GVL.arrValve_PM[0](in_out:= GVL.pm[0].inConv.valve[0]);
GVL.arrValve_PM[1](in_out:= GVL.pm[0].inConv.valve[1]);
GVL.arrValve_PM[2](in_out:= GVL.pm[0].inConv.valve[2]);
GVL.arrValve_PM[3](in_out:= GVL.pm[1].inConv.valve[0]);
GVL.arrValve_PM[4](in_out:= GVL.pm[1].inConv.valve[1]);
GVL.arrValve_PM[5](in_out:= GVL.pm[1].inConv.valve[2]);
GVL.arrValve_PM[6](in_out:= GVL.pm[2].inConv.valve[0]);
GVL.arrValve_PM[7](in_out:= GVL.pm[2].inConv.valve[1]);
GVL.arrValve_PM[8](in_out:= GVL.pm[2].inConv.valve[2]);
GVL.arrValve_PM[9](in_out:= GVL.pm[3].inConv.valve[0]);
GVL.arrValve_PM[10](in_out:= GVL.pm[3].inConv.valve[1]);
GVL.arrValve_PM[11](in_out:= GVL.pm[3].inConv.valve[2]);
GVL.arrValve_PM[12](in_out:= GVL.pm[4].inConv.valve[0]);
GVL.arrValve_PM[13](in_out:= GVL.pm[4].inConv.valve[1]);
GVL.arrValve_PM[14](in_out:= GVL.pm[4].inConv.valve[2]);
GVL.arrValve_PM[15](in_out:= GVL.pm[5].inConv.valve[0]);
GVL.arrValve_PM[16](in_out:= GVL.pm[5].inConv.valve[1]);
GVL.arrValve_PM[17](in_out:= GVL.pm[5].inConv.valve[2]);
GVL.arrValve_PM[18](in_out:= GVL.pm[6].inConv.valve[0]);
GVL.arrValve_PM[19](in_out:= GVL.pm[6].inConv.valve[1]);
GVL.arrValve_PM[20](in_out:= GVL.pm[6].inConv.valve[2]);
GVL.arrValve_PM[21](in_out:= GVL.pm[7].inConv.valve[0]);
GVL.arrValve_PM[22](in_out:= GVL.pm[7].inConv.valve[1]);
GVL.arrValve_PM[23](in_out:= GVL.pm[7].inConv.valve[2]);
GVL.arrValve_PM[24](in_out:= GVL.pm[8].inConv.valve[0]);
GVL.arrValve_PM[25](in_out:= GVL.pm[8].inConv.valve[1]);
GVL.arrValve_PM[26](in_out:= GVL.pm[8].inConv.valve[2]);
GVL.arrValve_PM[27](in_out:= GVL.pm[9].inConv.valve[0]);
GVL.arrValve_PM[28](in_out:= GVL.pm[9].inConv.valve[1]);
GVL.arrValve_PM[29](in_out:= GVL.pm[9].inConv.valve[2]);
GVL.arrValve_PM[30](in_out:= GVL.pm[0].outConv.valve[0]);
GVL.arrValve_PM[31](in_out:= GVL.pm[0].outConv.valve[1]);
GVL.arrValve_PM[32](in_out:= GVL.pm[1].outConv.valve[0]);
GVL.arrValve_PM[33](in_out:= GVL.pm[1].outConv.valve[1]);
GVL.arrValve_PM[34](in_out:= GVL.pm[2].outConv.valve[0]);
GVL.arrValve_PM[35](in_out:= GVL.pm[2].outConv.valve[1]);
GVL.arrValve_PM[36](in_out:= GVL.pm[3].outConv.valve[0]);
GVL.arrValve_PM[37](in_out:= GVL.pm[3].outConv.valve[1]);
GVL.arrValve_PM[38](in_out:= GVL.pm[4].outConv.valve[0]);
GVL.arrValve_PM[39](in_out:= GVL.pm[4].outConv.valve[1]);
GVL.arrValve_PM[40](in_out:= GVL.pm[5].outConv.valve[0]);
GVL.arrValve_PM[41](in_out:= GVL.pm[5].outConv.valve[1]);
GVL.arrValve_PM[42](in_out:= GVL.pm[6].outConv.valve[0]);
GVL.arrValve_PM[43](in_out:= GVL.pm[6].outConv.valve[1]);
GVL.arrValve_PM[44](in_out:= GVL.pm[7].outConv.valve[0]);
GVL.arrValve_PM[45](in_out:= GVL.pm[7].outConv.valve[1]);
GVL.arrValve_PM[46](in_out:= GVL.pm[8].outConv.valve[0]);
GVL.arrValve_PM[47](in_out:= GVL.pm[8].outConv.valve[1]);
GVL.arrValve_PM[48](in_out:= GVL.pm[9].outConv.valve[0]);
GVL.arrValve_PM[49](in_out:= GVL.pm[9].outConv.valve[1]);//end of pm
GVL.arrValve_PM[50](in_out:= GVL.lb[0].valve_stopper[0]);
GVL.arrValve_PM[51](in_out:= GVL.lb[0].valve_stopper[1]);
GVL.arrValve_PM[52](in_out:= GVL.lb[0].valve_stopper[2]);
GVL.arrValve_PM[53](in_out:= GVL.lb[0].valve_stopper[3]);
GVL.arrValve_PM[54](in_out:= GVL.lb[0].valve_stopper[4]);
GVL.arrValve_PM[55](in_out:= GVL.lb[0].valve_stopper[5]);
GVL.arrValve_PM[56](in_out:= GVL.lb[1].valve_stopper[0]);
GVL.arrValve_PM[57](in_out:= GVL.lb[1].valve_stopper[1]);
GVL.arrValve_PM[58](in_out:= GVL.lb[1].valve_stopper[2]);
GVL.arrValve_PM[59](in_out:= GVL.lb[1].valve_stopper[3]);
GVL.arrValve_PM[60](in_out:= GVL.lb[1].valve_stopper[4]);
GVL.arrValve_PM[61](in_out:= GVL.lb[1].valve_stopper[5]);//end of lb
GVL.arrValve_PM[62](in_out:= GVL.lc[0].valve_guide[0]);
GVL.arrValve_PM[63](in_out:= GVL.lc[0].valve_guide[1]);
GVL.arrValve_PM[64](in_out:= GVL.lc[0].valve_stopper[0]);
GVL.arrValve_PM[65](in_out:= GVL.lc[0].valve_stopper[1]);
GVL.arrValve_PM[66](in_out:= GVL.lc[0].lateral.valve_lift);
GVL.arrValve_PM[67](in_out:= GVL.lc[0].lateral.valve_clamp[0]);
GVL.arrValve_PM[68](in_out:= GVL.lc[0].lateral.valve_clamp[1]);
GVL.arrValve_PM[69](in_out:= GVL.lc[1].valve_guide[0]);
GVL.arrValve_PM[70](in_out:= GVL.lc[1].valve_guide[1]);
GVL.arrValve_PM[71](in_out:= GVL.lc[1].valve_stopper[0]);
GVL.arrValve_PM[72](in_out:= GVL.lc[1].valve_stopper[1]);
GVL.arrValve_PM[73](in_out:= GVL.lc[1].lateral.valve_lift);
GVL.arrValve_PM[74](in_out:= GVL.lc[1].lateral.valve_clamp[0]);
GVL.arrValve_PM[75](in_out:= GVL.lc[1].lateral.valve_clamp[1]);//end of lc
GVL.arrValve_PM[76](in_out:= GVL.fr[0].valve);
GVL.arrValve_PM[77](in_out:= GVL.fr[1].valve);//end of fr

//////////////////////////////////////REM/////////////////////////////////////
GVL.arrValve_Rem[0](in_out:= GVL.rem[0].infeed[0].valve_stopper);
GVL.arrValve_Rem[1](in_out:= GVL.rem[0].lift[0].valve_clamp);
GVL.arrValve_Rem[2](in_out:= GVL.rem[0].lift[0].valve_perturbation[0]);
GVL.arrValve_Rem[3](in_out:= GVL.rem[0].lift[0].valve_perturbation[1]);
GVL.arrValve_Rem[4](in_out:= GVL.rem[0].lift[0].valve_perturbation[2]);
GVL.arrValve_Rem[5](in_out:= GVL.rem[0].lift[0].valve_perturbation[3]);
GVL.arrValve_Rem[6](in_out:= GVL.rem[0].infeed[1].valve_stopper);
GVL.arrValve_Rem[7](in_out:= GVL.rem[0].lift[1].valve_clamp);
GVL.arrValve_Rem[8](in_out:= GVL.rem[0].lift[1].valve_perturbation[0]);
GVL.arrValve_Rem[9](in_out:= GVL.rem[0].lift[1].valve_perturbation[1]);
GVL.arrValve_Rem[10](in_out:= GVL.rem[0].lift[1].valve_perturbation[2]);
GVL.arrValve_Rem[11](in_out:= GVL.rem[0].lift[1].valve_perturbation[3]);
GVL.arrValve_Rem[12](in_out:= GVL.rem[1].infeed[0].valve_stopper);
GVL.arrValve_Rem[13](in_out:= GVL.rem[1].lift[0].valve_clamp);
GVL.arrValve_Rem[14](in_out:= GVL.rem[1].lift[0].valve_perturbation[0]);
GVL.arrValve_Rem[15](in_out:= GVL.rem[1].lift[0].valve_perturbation[1]);
GVL.arrValve_Rem[16](in_out:= GVL.rem[1].lift[0].valve_perturbation[2]);
GVL.arrValve_Rem[17](in_out:= GVL.rem[1].lift[0].valve_perturbation[3]);
GVL.arrValve_Rem[18](in_out:= GVL.rem[1].infeed[1].valve_stopper);
GVL.arrValve_Rem[19](in_out:= GVL.rem[1].lift[1].valve_clamp);
GVL.arrValve_Rem[20](in_out:= GVL.rem[1].lift[1].valve_perturbation[0]);
GVL.arrValve_Rem[21](in_out:= GVL.rem[1].lift[1].valve_perturbation[1]);
GVL.arrValve_Rem[22](in_out:= GVL.rem[1].lift[1].valve_perturbation[2]);
GVL.arrValve_Rem[23](in_out:= GVL.rem[1].lift[1].valve_perturbation[3]);
GVL.arrValve_Rem[24](in_out:= GVL.rem[2].infeed[0].valve_stopper);
GVL.arrValve_Rem[25](in_out:= GVL.rem[2].lift[0].valve_clamp);
GVL.arrValve_Rem[26](in_out:= GVL.rem[2].lift[0].valve_perturbation[0]);
GVL.arrValve_Rem[27](in_out:= GVL.rem[2].lift[0].valve_perturbation[1]);
GVL.arrValve_Rem[28](in_out:= GVL.rem[2].lift[0].valve_perturbation[2]);
GVL.arrValve_Rem[29](in_out:= GVL.rem[2].lift[0].valve_perturbation[3]);
GVL.arrValve_Rem[30](in_out:= GVL.rem[2].infeed[1].valve_stopper);
GVL.arrValve_Rem[31](in_out:= GVL.rem[2].lift[1].valve_clamp);
GVL.arrValve_Rem[32](in_out:= GVL.rem[2].lift[1].valve_perturbation[0]);
GVL.arrValve_Rem[33](in_out:= GVL.rem[2].lift[1].valve_perturbation[1]);
GVL.arrValve_Rem[34](in_out:= GVL.rem[2].lift[1].valve_perturbation[2]);
GVL.arrValve_Rem[35](in_out:= GVL.rem[2].lift[1].valve_perturbation[3]);
GVL.arrValve_Rem[36](in_out:= GVL.rem[3].infeed[0].valve_stopper);
GVL.arrValve_Rem[37](in_out:= GVL.rem[3].lift[0].valve_clamp);
GVL.arrValve_Rem[38](in_out:= GVL.rem[3].lift[0].valve_perturbation[0]);
GVL.arrValve_Rem[39](in_out:= GVL.rem[3].lift[0].valve_perturbation[1]);
GVL.arrValve_Rem[40](in_out:= GVL.rem[3].lift[0].valve_perturbation[2]);
GVL.arrValve_Rem[41](in_out:= GVL.rem[3].lift[0].valve_perturbation[3]);
GVL.arrValve_Rem[42](in_out:= GVL.rem[3].infeed[1].valve_stopper);
GVL.arrValve_Rem[43](in_out:= GVL.rem[3].lift[1].valve_clamp);
GVL.arrValve_Rem[44](in_out:= GVL.rem[3].lift[1].valve_perturbation[0]);
GVL.arrValve_Rem[45](in_out:= GVL.rem[3].lift[1].valve_perturbation[1]);
GVL.arrValve_Rem[46](in_out:= GVL.rem[3].lift[1].valve_perturbation[2]);
GVL.arrValve_Rem[47](in_out:= GVL.rem[3].lift[1].valve_perturbation[3]);
GVL.arrValve_Rem[48](in_out:= GVL.rem[4].infeed[0].valve_stopper);
GVL.arrValve_Rem[49](in_out:= GVL.rem[4].lift[0].valve_clamp);
GVL.arrValve_Rem[50](in_out:= GVL.rem[4].lift[0].valve_perturbation[0]);
GVL.arrValve_Rem[51](in_out:= GVL.rem[4].lift[0].valve_perturbation[1]);
GVL.arrValve_Rem[52](in_out:= GVL.rem[4].lift[0].valve_perturbation[2]);
GVL.arrValve_Rem[53](in_out:= GVL.rem[4].lift[0].valve_perturbation[3]);
GVL.arrValve_Rem[54](in_out:= GVL.rem[4].infeed[1].valve_stopper);
GVL.arrValve_Rem[55](in_out:= GVL.rem[4].lift[1].valve_clamp);
GVL.arrValve_Rem[56](in_out:= GVL.rem[4].lift[1].valve_perturbation[0]);
GVL.arrValve_Rem[57](in_out:= GVL.rem[4].lift[1].valve_perturbation[1]);
GVL.arrValve_Rem[58](in_out:= GVL.rem[4].lift[1].valve_perturbation[2]);
GVL.arrValve_Rem[59](in_out:= GVL.rem[4].lift[1].valve_perturbation[3]);
GVL.arrValve_Rem[60](in_out:= GVL.rem[5].infeed[0].valve_stopper);
GVL.arrValve_Rem[61](in_out:= GVL.rem[5].lift[0].valve_clamp);
GVL.arrValve_Rem[62](in_out:= GVL.rem[5].lift[0].valve_perturbation[0]);
GVL.arrValve_Rem[63](in_out:= GVL.rem[5].lift[0].valve_perturbation[1]);
GVL.arrValve_Rem[64](in_out:= GVL.rem[5].lift[0].valve_perturbation[2]);
GVL.arrValve_Rem[65](in_out:= GVL.rem[5].lift[0].valve_perturbation[3]);
GVL.arrValve_Rem[66](in_out:= GVL.rem[5].infeed[1].valve_stopper);
GVL.arrValve_Rem[67](in_out:= GVL.rem[5].lift[1].valve_clamp);
GVL.arrValve_Rem[68](in_out:= GVL.rem[5].lift[1].valve_perturbation[0]);
GVL.arrValve_Rem[69](in_out:= GVL.rem[5].lift[1].valve_perturbation[1]);
GVL.arrValve_Rem[70](in_out:= GVL.rem[5].lift[1].valve_perturbation[2]);
GVL.arrValve_Rem[71](in_out:= GVL.rem[5].lift[1].valve_perturbation[3]);
GVL.arrValve_Rem[72](in_out:= GVL.rem[6].infeed[0].valve_stopper);
GVL.arrValve_Rem[73](in_out:= GVL.rem[6].lift[0].valve_clamp);
GVL.arrValve_Rem[74](in_out:= GVL.rem[6].lift[0].valve_perturbation[0]);
GVL.arrValve_Rem[75](in_out:= GVL.rem[6].lift[0].valve_perturbation[1]);
GVL.arrValve_Rem[76](in_out:= GVL.rem[6].lift[0].valve_perturbation[2]);
GVL.arrValve_Rem[77](in_out:= GVL.rem[6].lift[0].valve_perturbation[3]);
GVL.arrValve_Rem[78](in_out:= GVL.rem[6].infeed[1].valve_stopper);
GVL.arrValve_Rem[79](in_out:= GVL.rem[6].lift[1].valve_clamp);
GVL.arrValve_Rem[80](in_out:= GVL.rem[6].lift[1].valve_perturbation[0]);
GVL.arrValve_Rem[81](in_out:= GVL.rem[6].lift[1].valve_perturbation[1]);
GVL.arrValve_Rem[82](in_out:= GVL.rem[6].lift[1].valve_perturbation[2]);
GVL.arrValve_Rem[83](in_out:= GVL.rem[6].lift[1].valve_perturbation[3]);
GVL.arrValve_Rem[84](in_out:= GVL.rem[7].infeed[0].valve_stopper);
GVL.arrValve_Rem[85](in_out:= GVL.rem[7].lift[0].valve_clamp);
GVL.arrValve_Rem[86](in_out:= GVL.rem[7].lift[0].valve_perturbation[0]);
GVL.arrValve_Rem[87](in_out:= GVL.rem[7].lift[0].valve_perturbation[1]);
GVL.arrValve_Rem[88](in_out:= GVL.rem[7].lift[0].valve_perturbation[2]);
GVL.arrValve_Rem[89](in_out:= GVL.rem[7].lift[0].valve_perturbation[3]);
GVL.arrValve_Rem[90](in_out:= GVL.rem[7].infeed[1].valve_stopper);
GVL.arrValve_Rem[91](in_out:= GVL.rem[7].lift[1].valve_clamp);
GVL.arrValve_Rem[92](in_out:= GVL.rem[7].lift[1].valve_perturbation[0]);
GVL.arrValve_Rem[93](in_out:= GVL.rem[7].lift[1].valve_perturbation[1]);
GVL.arrValve_Rem[94](in_out:= GVL.rem[7].lift[1].valve_perturbation[2]);
GVL.arrValve_Rem[95](in_out:= GVL.rem[7].lift[1].valve_perturbation[3]);
GVL.arrValve_Rem[96](in_out:= GVL.rem[8].infeed[0].valve_stopper);
GVL.arrValve_Rem[97](in_out:= GVL.rem[8].lift[0].valve_clamp);
GVL.arrValve_Rem[98](in_out:= GVL.rem[8].lift[0].valve_perturbation[0]);
GVL.arrValve_Rem[99](in_out:= GVL.rem[8].lift[0].valve_perturbation[1]);
GVL.arrValve_Rem[100](in_out:= GVL.rem[8].lift[0].valve_perturbation[2]);
GVL.arrValve_Rem[101](in_out:= GVL.rem[8].lift[0].valve_perturbation[3]);
GVL.arrValve_Rem[102](in_out:= GVL.rem[8].infeed[1].valve_stopper);
GVL.arrValve_Rem[103](in_out:= GVL.rem[8].lift[1].valve_clamp);
GVL.arrValve_Rem[104](in_out:= GVL.rem[8].lift[1].valve_perturbation[0]);
GVL.arrValve_Rem[105](in_out:= GVL.rem[8].lift[1].valve_perturbation[1]);
GVL.arrValve_Rem[106](in_out:= GVL.rem[8].lift[1].valve_perturbation[2]);
GVL.arrValve_Rem[107](in_out:= GVL.rem[8].lift[1].valve_perturbation[3]);
GVL.arrValve_Rem[108](in_out:= GVL.rem[9].infeed[0].valve_stopper);
GVL.arrValve_Rem[109](in_out:= GVL.rem[9].lift[0].valve_clamp);
GVL.arrValve_Rem[110](in_out:= GVL.rem[9].lift[0].valve_perturbation[0]);
GVL.arrValve_Rem[111](in_out:= GVL.rem[9].lift[0].valve_perturbation[1]);
GVL.arrValve_Rem[112](in_out:= GVL.rem[9].lift[0].valve_perturbation[2]);
GVL.arrValve_Rem[113](in_out:= GVL.rem[9].lift[0].valve_perturbation[3]);
GVL.arrValve_Rem[114](in_out:= GVL.rem[9].infeed[1].valve_stopper);
GVL.arrValve_Rem[115](in_out:= GVL.rem[9].lift[1].valve_clamp);
GVL.arrValve_Rem[116](in_out:= GVL.rem[9].lift[1].valve_perturbation[0]);
GVL.arrValve_Rem[117](in_out:= GVL.rem[9].lift[1].valve_perturbation[1]);
GVL.arrValve_Rem[118](in_out:= GVL.rem[9].lift[1].valve_perturbation[2]);
GVL.arrValve_Rem[119](in_out:= GVL.rem[9].lift[1].valve_perturbation[3]);
END_ACTION

METHOD M_ads_bagmachines : BOOL
VAR_INPUT
END_VAR
VAR
	
END_VAR
(*
ton_1ms(PT:=T#2MS);
FOR i:=0 TO 2 DO
	GVL.adsread[i](
				NETID:=GVL.netId_bagmachie[i] , 
				PORT:=851 , 
				IDXGRP:=16#00004020 , 
				IDXOFFS:=100 , 
				LEN:= SIZEOF(GVL.adsArr_bagMachine[i].inArr), 
				DESTADDR:= ADR(GVL.adsArr_bagMachine[i].inArr), 
				READ:=GVL.bread[i] , 
				TMOUT:=T#2S , 
				BUSY=> , 
				ERR=> , 
				ERRID=> );
	GVL.adswrite[i](
				NETID:=GVL.netId_bagmachie[i] , 
				PORT:=851, 
				IDXGRP:=16#00004020, 
				IDXOFFS:=200, 
				LEN:=SIZEOF(GVL.adsArr_bagMachine[i].outArr) , 
				SRCADDR:=ADR(GVL.adsArr_bagMachine[i].outArr) , 
				WRITE:=GVL.bwrite[i] , 
				TMOUT:=T#2S , 
				BUSY=> , 
				ERR=> , 
				ERRID=> );
		END_FOR
CASE iAds OF 
	0:
		FOR i:=0 TO 2 DO
			GVL.bread[i]	:=FALSE;
			GVL.bwrite[i]	:=FALSE;
		END_FOR
		iAds	:=1;
	1:
		ton_1ms.IN	:= TRUE;
		IF ton_1ms.Q THEN
			ton_1ms.IN	:= FALSE;
			iAds	:=2;
		END_IF
	2:
		FOR i:=0 TO 2 DO
			GVL.bread[i]	:=TRUE;
			GVL.bwrite[i]	:=TRUE;
		END_FOR
		iAds	:=3;
	3:
		ton_1ms.IN	:= TRUE;
		IF ton_1ms.Q THEN
			ton_1ms.IN	:= FALSE;
			iAds	:=0;
		END_IF		
END_CASE

*)
END_METHOD

METHOD M_agingTest : BOOL
VAR_INPUT
END_VAR
END_METHOD

METHOD M_checkError : BOOL
VAR_INPUT
END_VAR
VAR
	i	: INT;
END_VAR
M_checkError	:= FALSE;
xErr_converterMotors	:= FALSE;
FOR i:=0 TO 57 DO
	IF GVL.ref_fbconverterMotor[i]^.xErr THEN
		xErr_converterMotors	:= TRUE;
	END_IF
END_FOR
M_checkError	:= TRUE;
END_METHOD

METHOD M_mappingIO 
VAR_INPUT
END_VAR
////////////////////////////////////////////////////ReM////////////////////////////////////////////////////////////////
GVL.fb_remIOmapping[0](iReM:= 0);
GVL.fb_remIOmapping[1](iReM:= 1);
GVL.fb_remIOmapping[2](iReM:= 2);
GVL.fb_remIOmapping[3](iReM:= 3);
GVL.fb_remIOmapping[4](iReM:= 4);
GVL.fb_remIOmapping[5](iReM:= 5);
GVL.fb_remIOmapping[6](iReM:= 6);
GVL.fb_remIOmapping[7](iReM:= 7);
GVL.fb_remIOmapping[8](iReM:= 8);
GVL.fb_remIOmapping[9](iReM:= 9);
GVL.fb_remAxisMapping[0](iReM :=0,iLift:=0,sNetID:='192.168.11.159.4.1',nSlaveAddr:=1005);
GVL.fb_remAxisMapping[1](iReM :=0,iLift:=1,sNetID:='192.168.11.159.4.1',nSlaveAddr:=1006);
GVL.fb_remAxisMapping[2](iReM :=1,iLift:=0,sNetID:='192.168.11.159.4.1',nSlaveAddr:=1009);
GVL.fb_remAxisMapping[3](iReM :=1,iLift:=1,sNetID:='192.168.11.159.4.1',nSlaveAddr:=1010);
GVL.fb_remAxisMapping[4](iReM :=2,iLift:=0,sNetID:='192.168.11.159.4.1',nSlaveAddr:=1013);
GVL.fb_remAxisMapping[5](iReM :=2,iLift:=1,sNetID:='192.168.11.159.4.1',nSlaveAddr:=1014);
GVL.fb_remAxisMapping[6](iReM :=3,iLift:=0,sNetID:='192.168.11.159.4.1',nSlaveAddr:=1017);
GVL.fb_remAxisMapping[7](iReM :=3,iLift:=1,sNetID:='192.168.11.159.4.1',nSlaveAddr:=1018);
GVL.fb_remAxisMapping[8](iReM :=4,iLift:=0,sNetID:='192.168.11.159.4.1',nSlaveAddr:=1021);
GVL.fb_remAxisMapping[9](iReM :=4,iLift:=1,sNetID:='192.168.11.159.4.1',nSlaveAddr:=1022);
GVL.fb_remAxisMapping[10](iReM :=5,iLift:=0,sNetID:='192.168.11.159.4.1',nSlaveAddr:=1025);
GVL.fb_remAxisMapping[11](iReM :=5,iLift:=1,sNetID:='192.168.11.159.4.1',nSlaveAddr:=1026);
GVL.fb_remAxisMapping[12](iReM :=6,iLift:=0,sNetID:='192.168.11.159.4.1',nSlaveAddr:=1029);
GVL.fb_remAxisMapping[13](iReM :=6,iLift:=1,sNetID:='192.168.11.159.4.1',nSlaveAddr:=1030);
GVL.fb_remAxisMapping[14](iReM :=7,iLift:=0,sNetID:='192.168.11.159.4.1',nSlaveAddr:=1033);
GVL.fb_remAxisMapping[15](iReM :=7,iLift:=1,sNetID:='192.168.11.159.4.1',nSlaveAddr:=1034);
GVL.fb_remAxisMapping[16](iReM :=8,iLift:=0,sNetID:='192.168.11.159.4.1',nSlaveAddr:=1037);
GVL.fb_remAxisMapping[17](iReM :=8,iLift:=1,sNetID:='192.168.11.159.4.1',nSlaveAddr:=1038);
GVL.fb_remAxisMapping[18](iReM :=9,iLift:=0,sNetID:='192.168.11.159.4.1',nSlaveAddr:=1041);
GVL.fb_remAxisMapping[19](iReM :=9,iLift:=1,sNetID:='192.168.11.159.4.1',nSlaveAddr:=1042);
GVL.fbAxisCtrl_Lift[0](stAxisCtrl:=GVL.stAxisCtrl_Lift[0],IN_OUT:=GVL.rem[0].lift[0].st_mcAxis);
GVL.fbAxisCtrl_Lift[1](stAxisCtrl:=GVL.stAxisCtrl_Lift[1],IN_OUT:=GVL.rem[0].lift[1].st_mcAxis);
GVL.fbAxisCtrl_Lift[2](stAxisCtrl:=GVL.stAxisCtrl_Lift[2],IN_OUT:=GVL.rem[1].lift[0].st_mcAxis);
GVL.fbAxisCtrl_Lift[3](stAxisCtrl:=GVL.stAxisCtrl_Lift[3],IN_OUT:=GVL.rem[1].lift[1].st_mcAxis);
GVL.fbAxisCtrl_Lift[4](stAxisCtrl:=GVL.stAxisCtrl_Lift[4],IN_OUT:=GVL.rem[2].lift[0].st_mcAxis);
GVL.fbAxisCtrl_Lift[5](stAxisCtrl:=GVL.stAxisCtrl_Lift[5],IN_OUT:=GVL.rem[2].lift[1].st_mcAxis);
GVL.fbAxisCtrl_Lift[6](stAxisCtrl:=GVL.stAxisCtrl_Lift[6],IN_OUT:=GVL.rem[3].lift[0].st_mcAxis);
GVL.fbAxisCtrl_Lift[7](stAxisCtrl:=GVL.stAxisCtrl_Lift[7],IN_OUT:=GVL.rem[3].lift[1].st_mcAxis);
GVL.fbAxisCtrl_Lift[8](stAxisCtrl:=GVL.stAxisCtrl_Lift[8],IN_OUT:=GVL.rem[4].lift[0].st_mcAxis);
GVL.fbAxisCtrl_Lift[9](stAxisCtrl:=GVL.stAxisCtrl_Lift[9],IN_OUT:=GVL.rem[4].lift[1].st_mcAxis);
GVL.fbAxisCtrl_Lift[10](stAxisCtrl:=GVL.stAxisCtrl_Lift[10],IN_OUT:=GVL.rem[5].lift[0].st_mcAxis);
GVL.fbAxisCtrl_Lift[11](stAxisCtrl:=GVL.stAxisCtrl_Lift[11],IN_OUT:=GVL.rem[5].lift[1].st_mcAxis);
GVL.fbAxisCtrl_Lift[12](stAxisCtrl:=GVL.stAxisCtrl_Lift[12],IN_OUT:=GVL.rem[6].lift[0].st_mcAxis);
GVL.fbAxisCtrl_Lift[13](stAxisCtrl:=GVL.stAxisCtrl_Lift[13],IN_OUT:=GVL.rem[6].lift[1].st_mcAxis);
GVL.fbAxisCtrl_Lift[14](stAxisCtrl:=GVL.stAxisCtrl_Lift[14],IN_OUT:=GVL.rem[7].lift[0].st_mcAxis);
GVL.fbAxisCtrl_Lift[15](stAxisCtrl:=GVL.stAxisCtrl_Lift[15],IN_OUT:=GVL.rem[7].lift[1].st_mcAxis);
GVL.fbAxisCtrl_Lift[16](stAxisCtrl:=GVL.stAxisCtrl_Lift[16],IN_OUT:=GVL.rem[8].lift[0].st_mcAxis);
GVL.fbAxisCtrl_Lift[17](stAxisCtrl:=GVL.stAxisCtrl_Lift[17],IN_OUT:=GVL.rem[8].lift[1].st_mcAxis);
GVL.fbAxisCtrl_Lift[18](stAxisCtrl:=GVL.stAxisCtrl_Lift[18],IN_OUT:=GVL.rem[9].lift[0].st_mcAxis);
GVL.fbAxisCtrl_Lift[19](stAxisCtrl:=GVL.stAxisCtrl_Lift[19],IN_OUT:=GVL.rem[9].lift[1].st_mcAxis);


////////////////////////////////////////////////////PM////////////////////////////////////////////////////////////////
GVL.fb_rmIOmapping[0](iRm:= 0);
GVL.fb_rmIOmapping[1](iRm:= 1);
GVL.fb_rmIOmapping[2](iRm:= 2);
GVL.fb_rmIOmapping[3](iRm:= 3);
GVL.fb_rmIOmapping[4](iRm:= 4);
GVL.fb_pmAxisMapping[0](iPM :=0,iBuffer:=0,sNetID:='192.168.11.159.5.1',nSlaveAddr:=1010);
GVL.fb_pmAxisMapping[1](iPM :=0,iBuffer:=1,sNetID:='192.168.11.159.5.1',nSlaveAddr:=1011);
GVL.fb_pmAxisMapping[2](iPM :=1,iBuffer:=0,sNetID:='192.168.11.159.5.1',nSlaveAddr:=1012);
GVL.fb_pmAxisMapping[3](iPM :=1,iBuffer:=1,sNetID:='192.168.11.159.5.1',nSlaveAddr:=1013);
GVL.fb_pmAxisMapping[4](iPM :=2,iBuffer:=0,sNetID:='192.168.11.159.5.1',nSlaveAddr:=1020);
GVL.fb_pmAxisMapping[5](iPM :=2,iBuffer:=1,sNetID:='192.168.11.159.5.1',nSlaveAddr:=1021);
GVL.fb_pmAxisMapping[6](iPM :=3,iBuffer:=0,sNetID:='192.168.11.159.5.1',nSlaveAddr:=1022);
GVL.fb_pmAxisMapping[7](iPM :=3,iBuffer:=1,sNetID:='192.168.11.159.5.1',nSlaveAddr:=1023);
GVL.fb_pmAxisMapping[8](iPM :=4,iBuffer:=0,sNetID:='192.168.11.159.5.1',nSlaveAddr:=1028);
GVL.fb_pmAxisMapping[9](iPM :=4,iBuffer:=1,sNetID:='192.168.11.159.5.1',nSlaveAddr:=1029);
GVL.fb_pmAxisMapping[10](iPM :=5,iBuffer:=0,sNetID:='192.168.11.159.5.1',nSlaveAddr:=1030);
GVL.fb_pmAxisMapping[11](iPM :=5,iBuffer:=1,sNetID:='192.168.11.159.5.1',nSlaveAddr:=1031);
GVL.fb_pmAxisMapping[12](iPM :=6,iBuffer:=0,sNetID:='192.168.11.159.5.1',nSlaveAddr:=1036);
GVL.fb_pmAxisMapping[13](iPM :=6,iBuffer:=1,sNetID:='192.168.11.159.5.1',nSlaveAddr:=1037);
GVL.fb_pmAxisMapping[14](iPM :=7,iBuffer:=0,sNetID:='192.168.11.159.5.1',nSlaveAddr:=1038);
GVL.fb_pmAxisMapping[15](iPM :=7,iBuffer:=1,sNetID:='192.168.11.159.5.1',nSlaveAddr:=1039);
GVL.fb_pmAxisMapping[16](iPM :=8,iBuffer:=0,sNetID:='192.168.11.159.5.1',nSlaveAddr:=1046);
GVL.fb_pmAxisMapping[17](iPM :=8,iBuffer:=1,sNetID:='192.168.11.159.5.1',nSlaveAddr:=1047);
GVL.fb_pmAxisMapping[18](iPM :=9,iBuffer:=0,sNetID:='192.168.11.159.5.1',nSlaveAddr:=1048);
GVL.fb_pmAxisMapping[19](iPM :=9,iBuffer:=1,sNetID:='192.168.11.159.5.1',nSlaveAddr:=1049);

GVL.fbAxisCtrl_Buffer[0](stAxisCtrl:=GVL.stAxisCtrl_Buffer[0],IN_OUT:=GVL.pm[0].buffer[0].st_mcAxis);
GVL.fbAxisCtrl_Buffer[1](stAxisCtrl:=GVL.stAxisCtrl_Buffer[1],IN_OUT:=GVL.pm[0].buffer[1].st_mcAxis);
GVL.fbAxisCtrl_Buffer[2](stAxisCtrl:=GVL.stAxisCtrl_Buffer[2],IN_OUT:=GVL.pm[1].buffer[0].st_mcAxis);
GVL.fbAxisCtrl_Buffer[3](stAxisCtrl:=GVL.stAxisCtrl_Buffer[3],IN_OUT:=GVL.pm[1].buffer[1].st_mcAxis);
GVL.fbAxisCtrl_Buffer[4](stAxisCtrl:=GVL.stAxisCtrl_Buffer[4],IN_OUT:=GVL.pm[2].buffer[0].st_mcAxis);
GVL.fbAxisCtrl_Buffer[5](stAxisCtrl:=GVL.stAxisCtrl_Buffer[5],IN_OUT:=GVL.pm[2].buffer[1].st_mcAxis);
GVL.fbAxisCtrl_Buffer[6](stAxisCtrl:=GVL.stAxisCtrl_Buffer[6],IN_OUT:=GVL.pm[3].buffer[0].st_mcAxis);
GVL.fbAxisCtrl_Buffer[7](stAxisCtrl:=GVL.stAxisCtrl_Buffer[7],IN_OUT:=GVL.pm[3].buffer[1].st_mcAxis);
GVL.fbAxisCtrl_Buffer[8](stAxisCtrl:=GVL.stAxisCtrl_Buffer[8],IN_OUT:=GVL.pm[4].buffer[0].st_mcAxis);
GVL.fbAxisCtrl_Buffer[9](stAxisCtrl:=GVL.stAxisCtrl_Buffer[9],IN_OUT:=GVL.pm[4].buffer[1].st_mcAxis);
GVL.fbAxisCtrl_Buffer[10](stAxisCtrl:=GVL.stAxisCtrl_Buffer[10],IN_OUT:=GVL.pm[5].buffer[0].st_mcAxis);
GVL.fbAxisCtrl_Buffer[11](stAxisCtrl:=GVL.stAxisCtrl_Buffer[11],IN_OUT:=GVL.pm[5].buffer[1].st_mcAxis);
GVL.fbAxisCtrl_Buffer[12](stAxisCtrl:=GVL.stAxisCtrl_Buffer[12],IN_OUT:=GVL.pm[6].buffer[0].st_mcAxis);
GVL.fbAxisCtrl_Buffer[13](stAxisCtrl:=GVL.stAxisCtrl_Buffer[13],IN_OUT:=GVL.pm[6].buffer[1].st_mcAxis);
GVL.fbAxisCtrl_Buffer[14](stAxisCtrl:=GVL.stAxisCtrl_Buffer[14],IN_OUT:=GVL.pm[7].buffer[0].st_mcAxis);
GVL.fbAxisCtrl_Buffer[15](stAxisCtrl:=GVL.stAxisCtrl_Buffer[15],IN_OUT:=GVL.pm[7].buffer[1].st_mcAxis);
GVL.fbAxisCtrl_Buffer[16](stAxisCtrl:=GVL.stAxisCtrl_Buffer[16],IN_OUT:=GVL.pm[8].buffer[0].st_mcAxis);
GVL.fbAxisCtrl_Buffer[17](stAxisCtrl:=GVL.stAxisCtrl_Buffer[17],IN_OUT:=GVL.pm[8].buffer[1].st_mcAxis);
GVL.fbAxisCtrl_Buffer[18](stAxisCtrl:=GVL.stAxisCtrl_Buffer[18],IN_OUT:=GVL.pm[9].buffer[0].st_mcAxis);
GVL.fbAxisCtrl_Buffer[19](stAxisCtrl:=GVL.stAxisCtrl_Buffer[19],IN_OUT:=GVL.pm[9].buffer[1].st_mcAxis);


////////////////////////////////////////////////////LC&LB&FR////////////////////////////////////////////////////////////////
GVL.fb_lcIOmappiing[0](iLc:= 0,mcAxis:=GVL.lc[0].lateral.mcAxis,IN_OUT:=GVL.lc[0].lateral.st_mcAxis,nSlaveAddr:=1006,sNetID:='192.168.11.159.5.1');
GVL.fb_lcIOmappiing[1](iLc:= 1,mcAxis:=GVL.lc[1].lateral.mcAxis,IN_OUT:=GVL.lc[1].lateral.st_mcAxis,nSlaveAddr:=1055,sNetID:='192.168.11.159.5.1');
GVL.fbAxisCtrl_LC[0](stAxisCtrl:=GVL.stAxisCtrl_LC[0],IN_OUT:=GVL.lc[0].lateral.st_mcAxis);
GVL.fbAxisCtrl_LC[1](stAxisCtrl:=GVL.stAxisCtrl_LC[1],IN_OUT:=GVL.lc[1].lateral.st_mcAxis);
GVL.fb_lbIOmappiing[0](iLb:=0);
GVL.fb_lbIOmappiing[1](iLb:=1);
GVL.fb_frIOmappiing[0](iFR:= 0,mcAxis:=GVL.fr[0].mcAxis,IN_OUT:=GVL.fr[0].st_mcAxis,nSlaveAddr:=1016,sNetID:='192.168.11.159.5.1');
GVL.fb_frIOmappiing[1](iFR:= 1,mcAxis:=GVL.fr[1].mcAxis,IN_OUT:=GVL.fr[1].st_mcAxis,nSlaveAddr:=1042,sNetID:='192.168.11.159.5.1');
GVL.fbAxisCtrl_FR[0](stAxisCtrl:=GVL.stAxisCtrl_FR[0],IN_OUT:=GVL.fr[0].st_mcAxis);
GVL.fbAxisCtrl_FR[1](stAxisCtrl:=GVL.stAxisCtrl_FR[1],IN_OUT:=GVL.fr[1].st_mcAxis);
END_METHOD

METHOD M_measuringLC : BOOL
VAR_INPUT
END_VAR

VAR
	i: INT;
	j: INT;
END_VAR

//IF Process Data In(BYTE1!=0) try Process Data Out(BYTE0=64:Teach-in)
FOR i :=1 TO 32 DO
	GVL.ibyteNum[i] := i;
END_FOR
FOR i:=1 TO 32 DO	
	GVL.stMeasuringLC.arByte[i].Ch[0]	:= GVL.byteLC[i].0;
	GVL.stMeasuringLC.arByte[i].Ch[1]	:= GVL.byteLC[i].1;
	GVL.stMeasuringLC.arByte[i].Ch[2]	:= GVL.byteLC[i].2;
	GVL.stMeasuringLC.arByte[i].Ch[3]	:= GVL.byteLC[i].3;
	GVL.stMeasuringLC.arByte[i].Ch[4]	:= GVL.byteLC[i].4;
	GVL.stMeasuringLC.arByte[i].Ch[5]	:= GVL.byteLC[i].5;
	GVL.stMeasuringLC.arByte[i].Ch[6]	:= GVL.byteLC[i].6;
	GVL.stMeasuringLC.arByte[i].Ch[7]	:= GVL.byteLC[i].7;
END_FOR


GVL.stByte REF= GVL.stMeasuringLC;
END_METHOD

METHOD M_ReM : BOOL
VAR_INPUT
END_VAR

//========== Lift0 Axis Config ==========
(*GVL.rem[0].lift[0].mcAxis
(
	ZSN		:= GVL.rem[0].lift[0].limit_sensor[2] OR GVL.rem[0].lift[0].st_mcAxis.xHoming,
	ZSP		:= GVL.rem[0].lift[0].limit_sensor[1]	OR GVL.rem[0].lift[0].st_mcAxis.xHoming,
	IN_OUT	:= GVL.rem[0].lift[0].st_mcAxis, 
	AXIS	:= GVL.rem[0].lift[0].Axisref, 
);
GVL.rem[0].lift[0].st_mcAxis.bPosSensorShow	:= TRUE;
GVL.rem[0].lift[0].st_mcAxis.bNegSensorShow	:= TRUE;
GVL.rem[0].lift[0].st_mcAxis.bStopButtonShow	:= TRUE;
GVL.rem[0].lift[0].st_mcAxis.rMaxAcceleration	:= 50000;
GVL.rem[0].lift[0].st_mcAxis.rMaxDeceleration	:= 50000;
GVL.rem[0].lift[0].st_mcAxis.rMaxJerk			:= 500000;
GVL.rem[0].lift[0].st_mcAxis.rAcceleration	:= 2500;
GVL.rem[0].lift[0].st_mcAxis.rDeceleration	:= 2500;
GVL.rem[0].lift[0].st_mcAxis.rJerk			:= 12500;
GVL.rem[0].lift[0].st_mcAxis.rMaxVelocity		:= 100;
GVL.rem[0].lift[0].st_mcAxis.rMaxDistance		:= 50;
GVL.rem[0].lift[0].st_mcAxis.bPosSen	:= GVL.rem[0].lift[0].limit_sensor[1] ;
GVL.rem[0].lift[0].st_mcAxis.bNegSen	:= GVL.rem[0].lift[0].limit_sensor[2] ;
GVL.rem[0].lift[0].st_mcAxis.mcHome.bCalibrationCam	:= GVL.rem[0].lift[0].limit_sensor[0];
GVL.rem[0].lift[0].st_mcAxis.bPositionSensor	:= GVL.rem[0].lift[0].limit_sensor[0];
GVL.rem[0].lift[0].st_mcAxis.bdirFW	:= TRUE;
GVL.rem[0].lift[0].st_mcAxis.rSetPos	:= 0;
GVL.rem[0].lift[0].st_mcAxis.sNetID := '192.168.11.159.1.1';
GVL.rem[0].lift[0].st_mcAxis.nSlaveAddr	:= 1002;
//GVL.rem[0].lift[0].st_mcAxis.nSubIndex := 16#1F;
//GVL.rem[0].lift[0].st_mcAxis.nIndex	:= 16#2005;


//========== Lift1 Axis Config ==========
GVL.rem[0].lift[1].mcAxis
(
	ZSN		:= GVL.rem[0].lift[1].limit_sensor[2] OR GVL.rem[0].lift[1].st_mcAxis.xHoming,
	ZSP		:= GVL.rem[0].lift[1].limit_sensor[1]	OR GVL.rem[0].lift[1].st_mcAxis.xHoming,
	IN_OUT	:= GVL.rem[0].lift[1].st_mcAxis, 
	AXIS	:= GVL.rem[0].lift[1].Axisref, 
);
GVL.rem[0].lift[1].st_mcAxis.bPosSensorShow	:= TRUE;
GVL.rem[0].lift[1].st_mcAxis.bNegSensorShow	:= TRUE;
GVL.rem[0].lift[1].st_mcAxis.bStopButtonShow	:= TRUE;
GVL.rem[0].lift[1].st_mcAxis.rMaxAcceleration	:= 50000;
GVL.rem[0].lift[1].st_mcAxis.rMaxDeceleration	:= 50000;
GVL.rem[0].lift[1].st_mcAxis.rMaxJerk			:= 500000;
GVL.rem[0].lift[1].st_mcAxis.rAcceleration	:= 2500;
GVL.rem[0].lift[1].st_mcAxis.rDeceleration	:= 2500;
GVL.rem[0].lift[1].st_mcAxis.rJerk			:= 12500;
GVL.rem[0].lift[1].st_mcAxis.rMaxVelocity		:= 100;
GVL.rem[0].lift[1].st_mcAxis.rMaxDistance		:= 50;
GVL.rem[0].lift[1].st_mcAxis.bPosSen	:= GVL.rem[0].lift[1].limit_sensor[1] ;
GVL.rem[0].lift[1].st_mcAxis.bNegSen	:= GVL.rem[0].lift[1].limit_sensor[2] ;
GVL.rem[0].lift[1].st_mcAxis.mcHome.bCalibrationCam	:= GVL.rem[0].lift[1].limit_sensor[0];
GVL.rem[0].lift[1].st_mcAxis.bPositionSensor	:= GVL.rem[0].lift[1].limit_sensor[0];
GVL.rem[0].lift[1].st_mcAxis.bdirFW	:= TRUE;
GVL.rem[0].lift[1].st_mcAxis.rSetPos	:= 0;
GVL.rem[0].lift[1].st_mcAxis.sNetID := '192.168.11.159.1.1';
GVL.rem[0].lift[1].st_mcAxis.nSlaveAddr	:= 1003;
//GVL.rem[0].lift[1].st_mcAxis.nSubIndex := 16#1F;
//GVL.rem[0].lift[1].st_mcAxis.nIndex	:=  16#2005;

CASE GVL.iFRtest OF 
	0:		
		//IF GVL.rem[0].lift[0].st_mcAxis.xHomingDone THEN
			IF GVL.bTs1 THEN
				GVL.rem[0].lift[0].st_mcAxis.mcMoveAbsolute.Execute := FALSE;
				GVL.iFRtest :=1;
			END_IF
		//END_IF
	1://open positon
		GVL.rem[0].lift[0].st_mcAxis.rActualPosSet := 0;
		GVL.rem[0].lift[0].st_mcAxis.rVelocitySet := 300;			
		GVL.rem[0].lift[0].st_mcAxis.mcMoveAbsolute.Execute := TRUE;
		GVL.rem[0].lift[1].st_mcAxis.rActualPosSet := 0;
		GVL.rem[0].lift[1].st_mcAxis.rVelocitySet := 300;			
		GVL.rem[0].lift[1].st_mcAxis.mcMoveAbsolute.Execute := TRUE;
		IF GVL.rem[0].lift[0].st_mcAxis.mcMoveAbsolute.Done AND GVL.rem[0].lift[1].st_mcAxis.mcMoveAbsolute.Done THEN
			GVL.rem[0].lift[0].st_mcAxis.mcMoveAbsolute.Execute := FALSE;
			GVL.rem[0].lift[1].st_mcAxis.mcMoveAbsolute.Execute := FALSE;
			GVL.iFRtest := 2;
		END_IF
	
	2:
		ton_delay.IN := TRUE;
		IF ton_delay.Q THEN
			ton_delay.IN := FALSE;
			GVL.iFRtest := 3;
		END_IF
	3://close position
		GVL.rem[0].lift[0].st_mcAxis.rActualPosSet := 424;
		GVL.rem[0].lift[0].st_mcAxis.rVelocitySet := 300;			
		GVL.rem[0].lift[0].st_mcAxis.mcMoveAbsolute.Execute := TRUE;
		GVL.rem[0].lift[1].st_mcAxis.rActualPosSet := 424;
		GVL.rem[0].lift[1].st_mcAxis.rVelocitySet := 300;			
		GVL.rem[0].lift[1].st_mcAxis.mcMoveAbsolute.Execute := TRUE;		
		GVL.st_mcAxis[1].mcMoveAbsolute.Execute := TRUE;
			IF GVL.rem[0].lift[0].st_mcAxis.mcMoveAbsolute.Done AND GVL.rem[0].lift[1].st_mcAxis.mcMoveAbsolute.Done THEN
				GVL.rem[0].lift[0].st_mcAxis.mcMoveAbsolute.Execute := FALSE;
				GVL.rem[0].lift[1].st_mcAxis.mcMoveAbsolute.Execute := FALSE;
				GVL.iFRtest := 4;
			END_IF   
	4://delay
		ton_delay.IN := TRUE;
		IF ton_delay.Q THEN
			ton_delay.IN := FALSE;
			GVL.iFRtest := 5;
		END_IF
	5://open positon
		GVL.rem[0].lift[0].st_mcAxis.rActualPosSet := 0;
		GVL.rem[0].lift[0].st_mcAxis.rVelocitySet := 300;			
		GVL.rem[0].lift[0].st_mcAxis.mcMoveAbsolute.Execute := TRUE;
		GVL.rem[0].lift[1].st_mcAxis.rActualPosSet := 0;
		GVL.rem[0].lift[1].st_mcAxis.rVelocitySet := 300;			
		GVL.rem[0].lift[1].st_mcAxis.mcMoveAbsolute.Execute := TRUE;
		IF GVL.rem[0].lift[0].st_mcAxis.mcMoveAbsolute.Done AND GVL.rem[0].lift[1].st_mcAxis.mcMoveAbsolute.Done THEN
			GVL.rem[0].lift[0].st_mcAxis.mcMoveAbsolute.Execute := FALSE;
			GVL.rem[0].lift[1].st_mcAxis.mcMoveAbsolute.Execute := FALSE;
			GVL.iFRtest := 6;
		END_IF
	6:
		GVL.iFRtest := 0;
END_CASE*)
END_METHOD

METHOD M_reset : BOOL
VAR_INPUT

END_VAR

VAR
	i	: INT;
END_VAR

M_reset	:= FALSE;

CASE iReset OF
	0:
		iReset	:= 1;
	1:
		FOR i:=0 TO 57 DO
			GVL.ref_fbconverterMotor[i]^.reset	:= TRUE;
		END_FOR
		iReset	:=2;
	2:
		FOR i:=0 TO 57 DO
			GVL.ref_fbconverterMotor[i]^.reset	:= FALSE;
		END_FOR
		M_reset	:= TRUE;
		iReset	:=0;

END_CASE
END_METHOD

METHOD M_rfid : BOOL
VAR_INPUT
END_VAR

VAR
	i: INT;
	
END_VAR
byte1 := ASC(string1);
FOR i:=0 TO 3 DO	
	GVL.arIn[i].Ch[0]	:= GVL.rfidIn[i].0;
	GVL.arIn[i].Ch[1]	:= GVL.rfidIn[i].1;
	GVL.arIn[i].Ch[2]	:= GVL.rfidIn[i].2;
	GVL.arIn[i].Ch[3]	:= GVL.rfidIn[i].3;
	GVL.arIn[i].Ch[4]	:= GVL.rfidIn[i].4;
	GVL.arIn[i].Ch[5]	:= GVL.rfidIn[i].5;
	GVL.arIn[i].Ch[6]	:= GVL.rfidIn[i].6;
	GVL.arIn[i].Ch[7]	:= GVL.rfidIn[i].7;
	GVL.rfidOut[i].0	:= GVL.arOut[i].Ch[0];
	GVL.rfidOut[i].1	:= GVL.arOut[i].Ch[1];
	GVL.rfidOut[i].2	:= GVL.arOut[i].Ch[2];
	GVL.rfidOut[i].3	:= GVL.arOut[i].Ch[3];
	GVL.rfidOut[i].4	:= GVL.arOut[i].Ch[4];
	GVL.rfidOut[i].5	:= GVL.arOut[i].Ch[5];
	GVL.rfidOut[i].6	:= GVL.arOut[i].Ch[6];
	GVL.rfidOut[i].7	:= GVL.arOut[i].Ch[7];	
END_FOR

FOR i:=4 TO 31 DO
	GVL.rfidOut[i] := INT_TO_BYTE(28*GVL.n+i-3);
END_FOR
END_METHOD

METHOD runEveryCycle : BOOL
VAR_INPUT
END_VAR

VAR
	


END_VAR
(*
CASE GVL.iFRtest OF 
	0:		
		IF GVL.st_mcAxis[0].xHomingDone THEN
			IF GVL.bTs1 THEN
				GVL.st_mcAxis[0].mcMoveAbsolute.Execute := FALSE;
				GVL.iFRtest :=1;
			END_IF
		END_IF
		IF GVL.bBeltTs THEN
			G_IO.arDI[5].Ch[2] := TRUE;
			G_IO.arDI[5].Ch[3] := TRUE;
			GVL.st_mcAxis[0].mcMoveAbsolute.Execute := FALSE;
			GVL.iFRtest :=100;
		END_IF
	100:
		GVL.st_mcAxis[0].rActualPosSet := 60000000;
		GVL.st_mcAxis[0].rVelocitySet := 150;	
		GVL.st_mcAxis[0].mcMoveAbsolute.Execute := TRUE;	
		IF NOT GVL.bBeltTs THEN
			GVL.st_mcAxis[0].mcMoveAbsolute.Execute := FALSE;
			GVL.st_mcAxis[0].mcStop.Execute := TRUE;
			IF GVL.st_mcAxis[0].mcStop.Done THEN
				GVL.st_mcAxis[0].mcStop.Execute := FALSE;
				GVL.iFRtest :=0;
			END_IF
			
		END_IF
	1://open positon
		valve := FALSE;
		IF retracted THEN
			GVL.st_mcAxis[0].rActualPosSet := 102.8;
			GVL.st_mcAxis[0].rVelocitySet := 300;			
			GVL.st_mcAxis[0].mcMoveAbsolute.Execute := TRUE;
			IF GVL.st_mcAxis[0].mcMoveAbsolute.Done THEN
				GVL.st_mcAxis[0].mcMoveAbsolute.Execute := FALSE;
				GVL.iFRtest := 2;
			END_IF
		END_IF
	2://valve extend
		valve := TRUE;
		IF extended THEN
			GVL.iFRtest := 3;
		END_IF
	3://delay
		ton_delay.IN := TRUE;
		IF ton_delay.Q THEN
			ton_delay.IN := FALSE;
			GVL.iFRtest := 4;
		END_IF
	4://close position
		GVL.st_mcAxis[0].rActualPosSet := -78.4;
		GVL.st_mcAxis[0].rVelocitySet := 300;			
		GVL.st_mcAxis[0].mcMoveAbsolute.Execute := TRUE;
		IF GVL.st_mcAxis[0].mcMoveAbsolute.Done THEN
			GVL.st_mcAxis[0].mcMoveAbsolute.Execute := FALSE;
			GVL.iFRtest := 6;
		END_IF	   
	5://delay
		ton_delay.IN := TRUE;
		IF ton_delay.Q THEN
			ton_delay.IN := FALSE;
			GVL.iFRtest := 6;
		END_IF
	6://valve retract
		valve := FALSE;
		IF retracted THEN
			GVL.iFRtest := 7;
		END_IF	
	7://valve extend
		valve := TRUE;
		IF extended THEN
			GVL.iFRtest := 8;
		END_IF	
	8://delay
		ton_delay.IN := TRUE;
		IF ton_delay.Q THEN
			ton_delay.IN := FALSE;
			GVL.iFRtest := 9;
		END_IF
	9://open positon
		GVL.st_mcAxis[0].rActualPosSet := 102.8;
		GVL.st_mcAxis[0].rVelocitySet := 300;			
		GVL.st_mcAxis[0].mcMoveAbsolute.Execute := TRUE;
		IF GVL.st_mcAxis[0].mcMoveAbsolute.Done THEN
			GVL.st_mcAxis[0].mcMoveAbsolute.Execute := FALSE;
			GVL.iFRtest := 10;
		END_IF
	10:
		GVL.iFRtest := 0;
END_CASE
*)
END_METHOD

ACTION safetyConfig:
G_IO.arDO[95].Ch[2] := GVL.safetyin[28].0;//rst lamp
GVL.safetyOut[0].0	:= G_IO.arDI[95].Ch[2];//btn_rst
END_ACTION

END_PROGRAM

// ---- POUs/bagmachines/FB_BagOpener.TcPOU
FUNCTION_BLOCK FB_BagOpener
VAR_INPUT
  ams_net_id	: STRING;
END_VAR
VAR_OUTPUT
END_VAR
VAR
  	// Variable to be read from the app in python.
	status: BagMachineStatus;
  	bag_detection_status: BagDetectionStatus;
  	bag_holder_status: BagHolderStatus;
    bag_status: BagStatus;
	current_bag_cmd: BagCmd;
	current_bag_detection_cmd: BagDetectionCmd;

	adsread				: ADSREAD;
	adswrite			: ADSWRITE;
	iMethodTest			: BagMachineStatus;
	bagOpenStatus 		: BagMachineStatus;
  	error_code			: UINT;

	adsArr				: AdsArr;
	iState				: INT;
	iAds				: INT;
	ton_ms				: TON;
	iMachineStatus		: INT;//inArr[0]
	iBagStatus			: INT;//inArr[1]
	iBagDetectStatus	: INT;//inArr[2]
	//iBagCmd				: INT;//outArr[1]
	//iBagDetectCmd		: INT;//outArr[2]
	
	
	
END_VAR

	adsread(
			NETID:=ams_net_id , 
			PORT:=851 , 
			IDXGRP:=16#00004020 , 
			IDXOFFS:=100 , 
			LEN:= SIZEOF(adsArr.inArr), 
			DESTADDR:= ADR(adsArr.inArr), 
			READ:=, 
			TMOUT:=T#2S , 
			BUSY=> , 
			ERR=> , 
			ERRID=> );
	adswrite(
			NETID:=ams_net_id , 
			PORT:=851, 
			IDXGRP:=16#00004020, 
			IDXOFFS:=200, 
			LEN:=SIZEOF(adsArr.outArr) , 
			SRCADDR:=ADR(adsArr.outArr) , 
			WRITE:= , 
			TMOUT:=T#2S , 
			BUSY=> , 
			ERR=> , 
			ERRID=> );
ton_ms(PT:=T#2MS);			
CASE iAds OF 
	0:
		adsread.READ	:= FALSE;
		adswrite.WRITE	:= FALSE;	
		iAds	:=1;
	1:
		ton_ms.IN	:= TRUE;
		IF ton_ms.Q THEN
			ton_ms.IN	:= FALSE;
			iAds	:=2;
		END_IF
	2:
		adsread.READ	:= TRUE;
		adswrite.WRITE	:= TRUE;
		iAds	:=3;
	3:
		ton_ms.IN	:= TRUE;
		IF ton_ms.Q THEN
			ton_ms.IN	:= FALSE;
			iAds	:=0;
		END_IF	
END_CASE
//inputArr:
//		[0]:machine status;
//		[1]:bag status;
//		[2]:bag detect status(0:idle,1:ok,2:ng);	
//		[3]:fixture status
//outputArr:
//		[0]:line status;
//		[1]:bag cmd(0: do_nothing, 1:insert_bag, 2:bag_done_clamping);
//	    [2]:bag detect cmd(0:idle,1:trigger,2:reset);
iMachineStatus		:= WORD_TO_INT(adsArr.inArr[0]);
iBagStatus 			:= WORD_TO_INT(adsArr.inArr[1]);
iBagDetectStatus	:= WORD_TO_INT(adsArr.inArr[2]);

adsArr.outArr[1]	:= INT_TO_WORD(current_bag_cmd);
adsArr.outArr[2]	:= INT_TO_WORD(current_bag_detection_cmd);

CASE adsArr.inArr[0] OF
	0:status	:= BagMachineStatus.OFF;
	1:status	:= BagMachineStatus.BUSY;
	2:status	:= BagMachineStatus.READY;
	3:status	:= BagMachineStatus.RESET;
	4:status	:= BagMachineStatus.ERROR;
	5:status	:= BagMachineStatus.STOPPED;
END_CASE
CASE adsArr.inArr[1] OF
	0:bag_status	:= BagStatus.UNKNOWN;
	1:bag_status	:= BagStatus.READY;
	2:bag_status	:= BagStatus.INSERTED;
	3:bag_status	:= BagStatus.REMOVED;
END_CASE
CASE adsArr.inArr[2] OF
	0:bag_detection_status	:= BagDetectionStatus.UNKNOWN;
	1:bag_detection_status	:= BagDetectionStatus.OKAY;
	2:bag_detection_status	:= BagDetectionStatus.NG;
	3:bag_detection_status	:= BagDetectionStatus.ERROR;
END_CASE
CASE adsArr.inArr[3] OF
	0:bag_holder_status	:= BagHolderStatus.UNKNOWN;
	1:bag_holder_status	:= BagHolderStatus.DOWN;
	2:bag_holder_status	:= BagHolderStatus.UP;
END_CASE

CASE current_bag_detection_cmd OF
	BagDetectionCmd.DO_NOTHING:
		;
	BagDetectionCmd.GET_RESULT_FROM_CAMERA:
		IF get_result_from_camera() THEN
			current_bag_detection_cmd	:=0;
		END_IF		
	BagDetectionCmd.RESET_CAMERA:
		IF reset_camera() THEN
			current_bag_detection_cmd	:=0;
		END_IF	
END_CASE

CASE current_bag_cmd OF
	BagCmd.DO_NOTHING:
		;
	BagCmd.INSERT_BAG_HOLDER:
		IF fixture_ready() THEN
			current_bag_cmd	:=0;
		END_IF		
	BagCmd.REMOVE_BAG_HOLDER:
		IF bag_done_clamping() THEN
			current_bag_cmd	:=0;
		END_IF	
	BagCmd.STOP:
		current_bag_cmd	:= BagCmd.STOP;
		IF status = BagMachineStatus.STOPPED THEN
			current_bag_cmd	:= BagCmd.DO_NOTHING;
		END_IF
END_CASE

//test just for jdm to control io for testing bag machine easier

{attribute 'TcRpcEnable'}
METHOD PUBLIC bag_done_clamping : BOOL
VAR_INPUT
END_VAR
bag_done_clamping	:= FALSE;
current_bag_cmd	:= BagCmd.REMOVE_BAG_HOLDER;
IF bag_removed OR bag_ready THEN//avoid not catch signal of removed
	bag_done_clamping := TRUE;
	current_bag_cmd	:= BagCmd.DO_NOTHING;
END_IF
END_METHOD

PROPERTY bag_inserted : BOOL
GET
bag_inserted	:= (WORD_TO_INT(adsArr.inArr[1]) = BagStatus.INSERTED);
END_GET
END_PROPERTY

PROPERTY bag_ready : BOOL
GET
bag_ready	:= (WORD_TO_INT(adsArr.inArr[1])	= BagStatus.READY);
END_GET
END_PROPERTY

PROPERTY bag_removed : BOOL
GET
bag_removed	:= (WORD_TO_INT(adsArr.inArr[1])	= BagStatus.REMOVED);
END_GET
END_PROPERTY

{attribute 'TcRpcEnable'}
METHOD PUBLIC fixture_ready : BOOL
VAR_INPUT

END_VAR
fixture_ready	:= FALSE;
current_bag_cmd	:= BagCmd.INSERT_BAG_HOLDER;
IF bag_inserted THEN
	fixture_ready	:= TRUE;
	current_bag_cmd	:= 	BagCmd.DO_NOTHING;
END_IF
END_METHOD

{attribute 'TcRpcEnable'}
METHOD PUBLIC get_result_from_camera : BOOL
VAR_INPUT

END_VAR
get_result_from_camera	:= FALSE;

current_bag_detection_cmd := BagDetectionCmd.GET_RESULT_FROM_CAMERA;
IF iBagDetectStatus <> BagDetectionStatus.UNKNOWN THEN
	get_result_from_camera := TRUE;
	current_bag_detection_cmd := BagDetectionCmd.DO_NOTHING;
END_IF
END_METHOD

METHOD M_Init : BOOL
VAR_INPUT
END_VAR
M_Init	:= FALSE;
iState	:= BagMachineStatus.OFF;
current_bag_detection_cmd := BagDetectionCmd.DO_NOTHING;
current_bag_cmd	:= BagCmd.DO_NOTHING;
M_Init	:= TRUE;
END_METHOD

{attribute 'TcRpcEnable'}
METHOD PUBLIC reset_camera : BOOL
VAR_INPUT

END_VAR
reset_camera := FALSE;
current_bag_detection_cmd := BagDetectionCmd.RESET_CAMERA;
IF iBagDetectStatus = BagDetectionStatus.UNKNOWN THEN
	reset_camera := TRUE;
	current_bag_detection_cmd := BagDetectionCmd.DO_NOTHING;
END_IF
END_METHOD

END_FUNCTION_BLOCK

// ---- POUs/bagmachines/FB_BagCloser.TcPOU
FUNCTION_BLOCK FB_BagCloser
VAR_INPUT
  ams_net_id: STRING;
END_VAR
VAR_OUTPUT
END_VAR
VAR
	// Variable to be read from the app in python.
	status: BagMachineStatus;
	//bag_detection_status: BagDetectionStatus;
	bag_holder_status: BagHolderStatus;
	bag_status: BagStatus;
	current_bag_cmd: BagCmd;
	current_bag_height_status: BagHeightStatus;

	adsread				: ADSREAD;
	adswrite			: ADSWRITE;
	iMethodTest			: BagMachineStatus;
	bagCloseStatus 		: BagMachineStatus;
  	error_code			: UINT;

	adsArr				: AdsArr;
	iAds				: INT;
	ton_ms				: TON;

	iMachineStatus		: INT;//inArr[0]
	iBagStatus			: INT;//inArr[1]
	
	arr_fb_belt	: ARRAY[0..9] OF fb_interface_bagmachine;
END_VAR

	adsread(
			NETID:=ams_net_id , 
			PORT:=851 , 
			IDXGRP:=16#00004020 , 
			IDXOFFS:=100 , 
			LEN:= SIZEOF(adsArr.inArr), 
			DESTADDR:= ADR(adsArr.inArr), 
			READ:=, 
			TMOUT:=T#2S , 
			BUSY=> , 
			ERR=> , 
			ERRID=> );
	adswrite(
			NETID:=ams_net_id , 
			PORT:=851, 
			IDXGRP:=16#00004020, 
			IDXOFFS:=200, 
			LEN:=SIZEOF(adsArr.outArr) , 
			SRCADDR:=ADR(adsArr.outArr) , 
			WRITE:= , 
			TMOUT:=T#2S , 
			BUSY=> , 
			ERR=> , 
			ERRID=> );
ton_ms(PT:=T#2MS);			
CASE iAds OF 
	0:
		adsread.READ	:= FALSE;
		adswrite.WRITE	:= FALSE;	
		iAds	:=1;
	1:
		ton_ms.IN	:= TRUE;
		IF ton_ms.Q THEN
			ton_ms.IN	:= FALSE;
			iAds	:=2;
		END_IF
	2:
		adsread.READ	:= TRUE;
		adswrite.WRITE	:= TRUE;
		iAds	:=3;
	3:
		ton_ms.IN	:= TRUE;
		IF ton_ms.Q THEN
			ton_ms.IN	:= FALSE;
			iAds	:=0;
		END_IF	
END_CASE
//inputArr:
//		[0]:machine status;
//		[1]:bag status;
//		[2]:fixture status
//outputArr:
//		[0]:line status;
//		[1]:bag cmd(0: do_nothing, 1:take_bag,2:bag_done_unclamping;);
//		[2]:height detect cmd(0:idle,1:ok,2:ng)
iMachineStatus	:= WORD_TO_INT(adsArr.inArr[0]);
iBagStatus := WORD_TO_INT(adsArr.inArr[1]);
 
adsArr.outArr[1]	:= INT_TO_WORD(current_bag_cmd);
adsArr.outArr[2]	:= INT_TO_WORD(current_bag_height_status);

CASE adsArr.inArr[0] OF
	0:status	:= BagMachineStatus.OFF;
	1:status	:= BagMachineStatus.BUSY;
	2:status	:= BagMachineStatus.READY;
	3:status	:= BagMachineStatus.RESET;
	4:status	:= BagMachineStatus.ERROR;
	5:status	:= BagMachineStatus.STOPPED;
END_CASE
CASE adsArr.inArr[1] OF
	0:bag_status	:= BagStatus.UNKNOWN;
	1:bag_status	:= BagStatus.READY;
	2:bag_status	:= BagStatus.INSERTED;
	3:bag_status	:= BagStatus.REMOVED;
END_CASE
CASE adsArr.inArr[3] OF
	0:bag_holder_status	:= BagHolderStatus.UNKNOWN;
	1:bag_holder_status	:= BagHolderStatus.DOWN;
	2:bag_holder_status	:= BagHolderStatus.UP;
END_CASE


CASE current_bag_cmd OF
	BagCmd.DO_NOTHING:
		;
	BagCmd.INSERT_BAG_HOLDER:
		IF fixture_ready() THEN
			current_bag_cmd	:=0;
		END_IF		
	BagCmd.REMOVE_BAG_HOLDER:
		IF bag_done_unclamping() THEN
			current_bag_cmd	:=0;
		END_IF	
	BagCmd.STOP:
		current_bag_cmd	:= BagCmd.STOP;
		IF status = BagMachineStatus.STOPPED THEN
			current_bag_cmd	:= BagCmd.DO_NOTHING;
		END_IF
		
END_CASE


//
IF GVL.bBagmachine_test THEN
	arr_fb_belt[0](bRun:=adsArr.inArr[4].0,iPM:=1,iBelt:=1);
	arr_fb_belt[1](bRun:=adsArr.inArr[4].1,iPM:=1,iBelt:=0);
	arr_fb_belt[2](bRun:=adsArr.inArr[4].2,iPM:=2,iBelt:=1);
	arr_fb_belt[3](bRun:=adsArr.inArr[4].3,iPM:=2,iBelt:=0);
	arr_fb_belt[4](bRun:=adsArr.inArr[4].4,iPM:=3,iBelt:=1);
	arr_fb_belt[5](bRun:=adsArr.inArr[4].5,iPM:=3,iBelt:=0);
	arr_fb_belt[6](bRun:=adsArr.inArr[4].6,iPM:=4,iBelt:=1);
	arr_fb_belt[7](bRun:=adsArr.inArr[4].7,iPM:=4,iBelt:=0);
	arr_fb_belt[8](bRun:=adsArr.inArr[4].8,iPM:=5,iBelt:=1);
	arr_fb_belt[9](bRun:=adsArr.inArr[4].9,iPM:=5,iBelt:=0);
	GVL.pm[2].outConv.valve[1].retract	:= adsArr.inArr[5].0;
	GVL.pm[4].outConv.valve[1].retract	:= adsArr.inArr[5].1;
	G_IO.arDO[55].Ch[10] := adsArr.inArr[5].2;
	G_IO.arDO[55].Ch[11] := adsArr.inArr[5].3;
	G_IO.arDO[55].Ch[12] := adsArr.inArr[5].4;
	G_IO.arDO[55].Ch[13] := adsArr.inArr[5].5;
	G_IO.arDO[59].Ch[10] := adsArr.inArr[5].6;
	G_IO.arDO[59].Ch[11] := adsArr.inArr[5].7;
	G_IO.arDO[59].Ch[12] := adsArr.inArr[5].8;
	G_IO.arDO[59].Ch[13] := adsArr.inArr[5].9;
	
	adsArr.outArr[4].0	:= GVL.pm[2].outConv.photo_sensor[1];
	adsArr.outArr[4].1	:= GVL.pm[4].outConv.photo_sensor[1];
	adsArr.outArr[4].2	:= G_IO.arDI[77].Ch[0];
	adsArr.outArr[4].3	:= G_IO.arDI[77].Ch[1];
	adsArr.outArr[4].4	:= G_IO.arDI[77].Ch[4];
	adsArr.outArr[4].5	:= G_IO.arDI[77].Ch[5];
	adsArr.outArr[4].6	:= G_IO.arDI[78].Ch[0];
	adsArr.outArr[4].7	:= G_IO.arDI[78].Ch[1];
	adsArr.outArr[4].8	:= G_IO.arDI[78].Ch[4];
	adsArr.outArr[4].9	:= G_IO.arDI[78].Ch[5];
	
	
	
	
	
	GVL.pm[1].outConv.valve[1].retract	:= TRUE;
	GVL.pm[1].outConv.valve[0].retract	:= TRUE;
	//GVL.pm[2].outConv.valve[1].retract	:= TRUE;
	GVL.pm[2].outConv.valve[0].retract	:= TRUE	;
	GVL.pm[3].outConv.valve[1].retract	:= TRUE;
	GVL.pm[3].outConv.valve[0].retract	:= TRUE;
	//GVL.pm[4].outConv.valve[1].retract	:= TRUE;
	GVL.pm[4].outConv.valve[0].retract	:= TRUE;
	GVL.pm[5].outConv.valve[1].retract	:= TRUE;
	GVL.pm[5].outConv.valve[0].retract	:= TRUE;
	
END_IF

{attribute 'TcRpcEnable'}
METHOD PUBLIC bag_done_unclamping : BOOL
VAR_INPUT

END_VAR
bag_done_unclamping	:= FALSE;
current_bag_cmd	:= BagCmd.REMOVE_BAG_HOLDER;
IF bag_removed OR unload_ready THEN //avoid not catch signal of removed
	bag_done_unclamping := TRUE;
	current_bag_cmd	:= BagCmd.DO_NOTHING;
END_IF
END_METHOD

PROPERTY bag_removed : BOOL
GET
bag_removed	:= (WORD_TO_INT(adsArr.inArr[1])	= BagStatus.REMOVED);
END_GET
END_PROPERTY

{attribute 'TcRpcEnable'}
METHOD PUBLIC fixture_ready : BOOL
VAR_INPUT

END_VAR
fixture_ready	:= FALSE;
current_bag_cmd	:= BagCmd.INSERT_BAG_HOLDER;
IF machine_inserted THEN
	fixture_ready	:= TRUE;
	current_bag_cmd	:= 	BagCmd.DO_NOTHING;
END_IF
END_METHOD

METHOD M_Init : BOOL
VAR_INPUT
END_VAR
M_Init	:= FALSE;
current_bag_cmd	:= BagCmd.DO_NOTHING;
current_bag_height_status := BagHeightStatus.UNKNOWN;
M_Init	:= TRUE;
END_METHOD

PROPERTY machine_inserted : BOOL
GET
machine_inserted	:= (WORD_TO_INT(adsArr.inArr[1])	= BagStatus.INSERTED);
END_GET
END_PROPERTY

PROPERTY unload_ready : BOOL
GET
unload_ready	:= (WORD_TO_INT(adsArr.inArr[1])	= BagStatus.READY);
END_GET
END_PROPERTY

END_FUNCTION_BLOCK

// ---- POUs/bagmachines/fb_interface_bagmachine.TcPOU
FUNCTION_BLOCK fb_interface_bagmachine
VAR_INPUT
	bRun: BOOL;
	iPM	: INT;
	iBelt	: INT;
END_VAR
VAR_OUTPUT
END_VAR
VAR
END_VAR

IF bRun THEN
	GVL.pm[iPM].outConv.belt[iBelt].fbconverter.cmd	:= INT_TO_UINT(E_CMD_ConverterMotor.BACKWARE);
	GVL.pm[iPM].outConv.belt[iBelt].fbconverter.freq	:= 3500;	
ELSE
	GVL.pm[iPM].outConv.belt[iBelt].fbconverter.cmd	:= INT_TO_UINT(E_CMD_ConverterMotor.STOP);
	GVL.pm[iPM].outConv.belt[iBelt].fbconverter.freq	:= 0;
END_IF

END_FUNCTION_BLOCK

// ---- POUs/bagmachines/FB_BagCompactor.TcPOU
FUNCTION_BLOCK FB_BagCompactor
VAR_INPUT
  ams_net_id: STRING;
END_VAR
VAR_OUTPUT
END_VAR
VAR
  status: BagMachineStatus;
  error_code: UINT;
END_VAR

{attribute 'TcRpcEnable'}
METHOD PUBLIC compact_bag : BOOL
VAR_INPUT

END_VAR
END_METHOD

END_FUNCTION_BLOCK

// ---- POUs/FB_heightDetection.TcPOU
FUNCTION_BLOCK FB_heightDetection
VAR_INPUT
	
END_VAR
VAR_IN_OUT
	stHeightDetection	: ST_heightDetection;
END_VAR
VAR_OUTPUT
	
END_VAR
VAR
	coeWrt		:	FB_EcCoESdoWrite;
	coeRead		:  	FB_EcCoESdoRead;
	iState	: INT;
	ton_wait : TON;
	heightCmd	: E_HeightDetection;
	height_detection_cmd : E_HeightDetection;//for server to call the method
	iHeight	: DWORD;//0.01mm
END_VAR


coeWrt(
	sNetId:= stHeightDetection.sNetID, 
	nSlaveAddr:=stHeightDetection.nSlaveAddr, 
	nSubIndex:= stHeightDetection.nSubIndex, 
	nIndex:= stHeightDetection.nIndex, 
	pSrcBuf:= ADR(stHeightDetection.iSdoWrite), 
	cbBufLen:= SIZEOF(stHeightDetection.iSdoWrite), 
	bExecute:= , 
	tTimeout:= , 
	bBusy=> , 
	bError=> , 
	nErrId=> );
coeRead(
	sNetId:= stHeightDetection.sNetID, 
	nSlaveAddr:=stHeightDetection.nSlaveAddr, 
	nSubIndex:= stHeightDetection.nSubIndex, 
	nIndex:= stHeightDetection.nIndex, 
	pDstBuf:= ADR(stHeightDetection.iSdoRead), 
	cbBufLen:= SIZEOF(stHeightDetection.iSdoRead), 
	bExecute:= , 
	tTimeout:= , 
	bBusy=> , 
	bError=> , 
	nErrId=> );
ton_wait();
CASE height_detection_cmd OF
	E_HeightDetection.SET_PROGRAM:
		IF M_setProg(iProgram:=16#05) THEN
			height_detection_cmd:= E_HeightDetection.DO_NOTHING;
		END_IF
	E_HeightDetection.READ_HEIGHT:
		IF M_readHeight(iTool:=16#00) THEN
			height_detection_cmd:= E_HeightDetection.DO_NOTHING;
		END_IF	
END_CASE

METHOD M_readHeight : BOOL
VAR_INPUT
	iTool	: DWORD;
END_VAR
VAR_OUTPUT
	
END_VAR
M_readHeight	:= FALSE;
CASE iState OF
	0:
		coeWrt.bExecute	:= FALSE;
		coeRead.bExecute:= FALSE;
		ton_wait.IN	:= FALSE;
		iState	:= 1;
	1://trig
		stHeightDetection.nIndex	:= 16#8005;
		stHeightDetection.nSubIndex	:= 16#01;
		stHeightDetection.iSdoWrite	:= 16#01;
		coeWrt.bExecute	:= TRUE;
		ton_wait.IN	:= TRUE;
		ton_wait.PT:= T#2S;
		IF ton_wait.Q THEN//wait finish
			coeWrt.bExecute	:= FALSE;
			iState	:= 2;
		END_IF			
	2://read tool
		IF NOT coeWrt.bBusy THEN
			stHeightDetection.nIndex	:= 16#8005;
			stHeightDetection.nSubIndex	:= 16#0B;
			stHeightDetection.iSdoWrite	:= iTool;
			coeWrt.bExecute	:= TRUE;
			iState	:= 3;
		END_IF
	3:
		IF coeWrt.bBusy THEN
			coeWrt.bExecute:= FALSE;
			iState	:= 4;
		END_IF
	4://respose of read tool
		IF NOT coeWrt.bBusy THEN
			stHeightDetection.nIndex	:= 16#8005;
			stHeightDetection.nSubIndex	:= 16#0C;		
			coeRead.bExecute	:= TRUE;
			IF coeRead.bBusy THEN
				coeRead.bExecute:= FALSE;
				iState	:= 5;
			END_IF
		END_IF	
	5://read value
		IF NOT coeRead.bBusy THEN
			stHeightDetection.nIndex	:= 16#8005;
			stHeightDetection.nSubIndex	:= 16#0D;		
			coeRead.bExecute	:= TRUE;
			iState	:= 6;
		END_IF
	6:
		IF coeRead.bBusy THEN
			coeRead.bExecute:= FALSE;
			iState	:= 7;
		END_IF
	7:
		IF NOT coeRead.bBusy THEN
			iHeight	:= stHeightDetection.iSdoRead;		
			iState	:= 8;
		END_IF
	8://init trig
		stHeightDetection.nIndex	:= 16#8005;
		stHeightDetection.nSubIndex	:= 16#01;
		stHeightDetection.iSdoWrite	:= 16#00;
		coeWrt.bExecute	:= TRUE;
		IF coeWrt.bBusy THEN
			coeWrt.bExecute	:= FALSE;
			iState	:= 9;
		END_IF
	9:
		IF NOT coeWrt.bBusy THEN
			M_readHeight	:= TRUE;
			iState	:= 0;
		END_IF
				
END_CASE
END_METHOD

METHOD M_setProg : BOOL
VAR_INPUT
	iProgram	: DWORD;
END_VAR
M_setProg	:= FALSE;
CASE iState OF
	0:
		iState	:= 1;
	1:
		stHeightDetection.nIndex	:= 16#8005;
		stHeightDetection.nSubIndex	:= 16#03;
		stHeightDetection.iSdoWrite	:= iProgram;
		coeWrt.bExecute	:= TRUE;
		iState	:= 2;
	2:
		ton_wait.IN := TRUE;
		ton_wait.PT	:= T#1000MS;
		stHeightDetection.nIndex	:= 16#8005;
		stHeightDetection.nSubIndex	:= 16#04;		
		coeRead.bExecute	:= ton_wait.Q;
		IF stHeightDetection.iSdoRead = 1 THEN
			M_setProg	:= TRUE;
			iState	:= 0;
		END_IF
		
		
END_CASE
END_METHOD

END_FUNCTION_BLOCK

// ---- POUs/FB_remAxisMapping.TcPOU
FUNCTION_BLOCK FB_remAxisMapping
VAR_INPUT
	iReM	: INT;
	iLift	: INT;
	sNetID	: STRING;
	nSlaveAddr : UINT;
END_VAR
VAR_OUTPUT
END_VAR
VAR
END_VAR

//========== Axis Config ==========
GVL.rem[iReM].lift[iLift].mcAxis
(
	ZSN		:= GVL.rem[iReM].lift[iLift].limit_sensor[2] OR GVL.rem[iReM].lift[iLift].st_mcAxis.xHoming,
	ZSP		:= GVL.rem[iReM].lift[iLift].limit_sensor[1]	OR GVL.rem[iReM].lift[iLift].st_mcAxis.xHoming,
	IN_OUT	:= GVL.rem[iReM].lift[iLift].st_mcAxis, 
	AXIS	:= GVL.rem[iReM].lift[iLift].Axisref, 
);
GVL.rem[iReM].lift[iLift].st_mcAxis.bPosSensorShow	:= TRUE;
GVL.rem[iReM].lift[iLift].st_mcAxis.bNegSensorShow	:= TRUE;
GVL.rem[iReM].lift[iLift].st_mcAxis.bStopButtonShow	:= TRUE;
GVL.rem[iReM].lift[iLift].st_mcAxis.rMaxAcceleration	:= 50000;
GVL.rem[iReM].lift[iLift].st_mcAxis.rMaxDeceleration	:= 50000;
GVL.rem[iReM].lift[iLift].st_mcAxis.rMaxJerk			:= 500000;
GVL.rem[iReM].lift[iLift].st_mcAxis.rAcceleration	:= 2500;
GVL.rem[iReM].lift[iLift].st_mcAxis.rDeceleration	:= 2500;
GVL.rem[iReM].lift[iLift].st_mcAxis.rJerk			:= 12500;
GVL.rem[iReM].lift[iLift].st_mcAxis.rMaxVelocity		:= 100;
GVL.rem[iReM].lift[iLift].st_mcAxis.rMaxDistance		:= 50;
GVL.rem[iReM].lift[iLift].st_mcAxis.bPosSen	:= GVL.rem[iReM].lift[iLift].limit_sensor[1] ;
GVL.rem[iReM].lift[iLift].st_mcAxis.bNegSen	:= GVL.rem[iReM].lift[iLift].limit_sensor[2] ;
GVL.rem[iReM].lift[iLift].st_mcAxis.mcHome.bCalibrationCam	:= GVL.rem[iReM].lift[iLift].limit_sensor[0];
GVL.rem[iReM].lift[iLift].st_mcAxis.bPositionSensor	:= GVL.rem[iReM].lift[iLift].limit_sensor[0];
GVL.rem[iReM].lift[iLift].st_mcAxis.bdirFW	:= TRUE;
GVL.rem[iReM].lift[iLift].st_mcAxis.rSetPos	:= 0;
GVL.rem[iReM].lift[iLift].st_mcAxis.sNetID := sNetID;
GVL.rem[iReM].lift[iLift].st_mcAxis.nSlaveAddr	:= nSlaveAddr;

END_FUNCTION_BLOCK

// ---- POUs/FB_rmIOmapping.TcPOU
FUNCTION_BLOCK FB_rmIOmapping
VAR_INPUT
	iRm	: INT;
END_VAR
VAR_OUTPUT
END_VAR
	
VAR
	offsetIn	: INT;
	offsetOut	: INT;
	rTrig_power_inConv	: R_TRIG;
	fTrig_power_inConv	: F_TRIG;
	rTrig_power_outConv	: R_TRIG;
	fTrig_power_outConv	: F_TRIG;
	
END_VAR

offsetIn	:= 50+iRm*5;
offsetOut	:= 50+iRm*4;
//pm[odd]
GVL.pm[iRm*2].buffer[0].contractor_axis				:= G_IO.arDI[offsetIn].Ch[0];
GVL.pm[iRm*2].buffer[0].axis_sensor					:= G_IO.arDI[offsetIn].Ch[1];
GVL.pm[iRm*2].buffer[0].surfae_slot_0				:= G_IO.arDI[offsetIn].Ch[2];
GVL.pm[iRm*2].buffer[0].surfae_slot_1				:= G_IO.arDI[offsetIn].Ch[3];
GVL.pm[iRm*2].buffer[0].surfae_slot_2				:= G_IO.arDI[offsetIn].Ch[4];
GVL.pm[iRm*2].buffer[0].above_fixture_light_curtain	:= G_IO.arDI[offsetIn].Ch[5];
GVL.pm[iRm*2].buffer[0].button						:= G_IO.arDI[offsetIn].Ch[6];
GVL.pm[iRm*2].buffer[0].locked						:= G_IO.arDI[offsetIn].Ch[7];
GVL.pm[iRm*2].buffer[0].magnet_locked				:= G_IO.arDI[offsetIn].Ch[8];
GVL.pm[iRm*2].buffer[1].contractor_axis				:= G_IO.arDI[offsetIn].Ch[9];
GVL.pm[iRm*2].buffer[1].axis_sensor					:= G_IO.arDI[offsetIn].Ch[10];
GVL.pm[iRm*2].buffer[1].surfae_slot_0				:= G_IO.arDI[offsetIn].Ch[11];
GVL.pm[iRm*2].buffer[1].surfae_slot_1				:= G_IO.arDI[offsetIn].Ch[12];
GVL.pm[iRm*2].buffer[1].surfae_slot_2				:= G_IO.arDI[offsetIn].Ch[13];
GVL.pm[iRm*2].buffer[1].above_fixture_light_curtain	:= G_IO.arDI[offsetIn].Ch[14];
GVL.pm[iRm*2].buffer[1].button						:= G_IO.arDI[offsetIn].Ch[15];
GVL.pm[iRm*2].buffer[1].locked						:= G_IO.arDI[offsetIn+1].Ch[0];
GVL.pm[iRm*2].buffer[1].magnet_locked				:= G_IO.arDI[offsetIn+1].Ch[1];
GVL.pm[iRm*2].contactor_robot						:= G_IO.arDI[offsetIn+1].Ch[2];
GVL.pm[iRm*2].inConv.valve[0].extended				:= G_IO.arDI[offsetIn+1].Ch[3];
GVL.pm[iRm*2].inConv.valve[0].retracted				:= G_IO.arDI[offsetIn+1].Ch[4];
GVL.pm[iRm*2].inConv.valve[1].extended				:= G_IO.arDI[offsetIn+1].Ch[5];
GVL.pm[iRm*2].inConv.valve[1].retracted				:= G_IO.arDI[offsetIn+1].Ch[6];
GVL.pm[iRm*2].inConv.valve[2].extended				:= G_IO.arDI[offsetIn+1].Ch[7];
GVL.pm[iRm*2].inConv.valve[2].retracted				:= G_IO.arDI[offsetIn+1].Ch[8];
GVL.pm[iRm*2].outConv.photo_sensor[0]				:= G_IO.arDI[offsetIn+1].Ch[9];
GVL.pm[iRm*2].outConv.photo_sensor[1]				:= G_IO.arDI[offsetIn+1].Ch[10];
GVL.pm[iRm*2].outConv.valve[0].extended				:= G_IO.arDI[offsetIn+1].Ch[11];
GVL.pm[iRm*2].outConv.valve[0].retracted			:= G_IO.arDI[offsetIn+1].Ch[12];
GVL.pm[iRm*2].outConv.valve[1].extended				:= G_IO.arDI[offsetIn+1].Ch[13];
GVL.pm[iRm*2].outConv.valve[1].retracted			:= G_IO.arDI[offsetIn+1].Ch[14];
GVL.pm[iRm*2].inConv.photo_sensor[0]				:= G_IO.arDI[offsetIn+4].Ch[2];
GVL.pm[iRm*2].inConv.photo_sensor[1]				:= G_IO.arDI[offsetIn+4].Ch[3];
GVL.pm[iRm*2].inConv.photo_sensor[2]				:= G_IO.arDI[offsetIn+4].Ch[4];
GVL.pm[iRm*2].inConv.photo_sensor[3]				:= G_IO.arDI[offsetIn+4].Ch[5];
GVL.pm[iRm*2].inConv.photo_sensor[4]				:= G_IO.arDI[offsetIn+4].Ch[6];
GVL.pm[iRm*2].inConv.photo_sensor[5]				:= G_IO.arDI[offsetIn+4].Ch[7];




G_IO.arDO[offsetOut].Ch[0]	:= GVL.pm[iRm*2].buffer[0].power_axis;
G_IO.arDO[offsetOut].Ch[1]	:= GVL.pm[iRm*2].buffer[0].magnet;
G_IO.arDO[offsetOut].Ch[2]	:= GVL.pm[iRm*2].buffer[1].power_axis;
G_IO.arDO[offsetOut].Ch[3]	:= GVL.pm[iRm*2].buffer[1].magnet;
G_IO.arDO[offsetOut].Ch[4]	:= GVL.pm[iRm*2].power_robot;
G_IO.arDO[offsetOut].Ch[12]	:= GVL.pm[iRm*2].buffer[0].lamp_button;
G_IO.arDO[offsetOut].Ch[13]	:= GVL.pm[iRm*2].buffer[1].lamp_button;
	
G_IO.arDO[offsetOut+1].Ch[0]	:= GVL.pm[iRm*2].inConv.valve[0].retract;
G_IO.arDO[offsetOut+1].Ch[1]	:= GVL.pm[iRm*2].inConv.valve[1].retract;
G_IO.arDO[offsetOut+1].Ch[2]	:= GVL.pm[iRm*2].inConv.valve[2].retract;
G_IO.arDO[offsetOut+1].Ch[6]	:= GVL.pm[iRm*2].outConv.valve[0].retract;
G_IO.arDO[offsetOut+1].Ch[7]	:= GVL.pm[iRm*2].outConv.valve[1].retract;




//pm[even]
GVL.pm[iRm*2+1].buffer[0].contractor_axis				:= G_IO.arDI[offsetIn+2].Ch[0];
GVL.pm[iRm*2+1].buffer[0].axis_sensor					:= G_IO.arDI[offsetIn+2].Ch[1];
GVL.pm[iRm*2+1].buffer[0].surfae_slot_0				:= G_IO.arDI[offsetIn+2].Ch[2];
GVL.pm[iRm*2+1].buffer[0].surfae_slot_1				:= G_IO.arDI[offsetIn+2].Ch[3];
GVL.pm[iRm*2+1].buffer[0].surfae_slot_2				:= G_IO.arDI[offsetIn+2].Ch[4];
GVL.pm[iRm*2+1].buffer[0].above_fixture_light_curtain	:= G_IO.arDI[offsetIn+2].Ch[5];
GVL.pm[iRm*2+1].buffer[0].button						:= G_IO.arDI[offsetIn+2].Ch[6];
GVL.pm[iRm*2+1].buffer[0].locked						:= G_IO.arDI[offsetIn+2].Ch[7];
GVL.pm[iRm*2+1].buffer[0].magnet_locked				:= G_IO.arDI[offsetIn+2].Ch[8];
GVL.pm[iRm*2+1].buffer[1].contractor_axis				:= G_IO.arDI[offsetIn+2].Ch[9];
GVL.pm[iRm*2+1].buffer[1].axis_sensor					:= G_IO.arDI[offsetIn+2].Ch[10];
GVL.pm[iRm*2+1].buffer[1].surfae_slot_0				:= G_IO.arDI[offsetIn+2].Ch[11];
GVL.pm[iRm*2+1].buffer[1].surfae_slot_1				:= G_IO.arDI[offsetIn+2].Ch[12];
GVL.pm[iRm*2+1].buffer[1].surfae_slot_2				:= G_IO.arDI[offsetIn+2].Ch[13];
GVL.pm[iRm*2+1].buffer[1].above_fixture_light_curtain	:= G_IO.arDI[offsetIn+2].Ch[14];
GVL.pm[iRm*2+1].buffer[1].button						:= G_IO.arDI[offsetIn+2].Ch[15];
GVL.pm[iRm*2+1].buffer[1].locked						:= G_IO.arDI[offsetIn+3].Ch[0];
GVL.pm[iRm*2+1].buffer[1].magnet_locked				:= G_IO.arDI[offsetIn+3].Ch[1];
GVL.pm[iRm*2+1].contactor_robot						:= G_IO.arDI[offsetIn+3].Ch[2];
GVL.pm[iRm*2+1].inConv.valve[0].extended				:= G_IO.arDI[offsetIn+3].Ch[3];
GVL.pm[iRm*2+1].inConv.valve[0].retracted				:= G_IO.arDI[offsetIn+3].Ch[4];
GVL.pm[iRm*2+1].inConv.valve[1].extended				:= G_IO.arDI[offsetIn+3].Ch[5];
GVL.pm[iRm*2+1].inConv.valve[1].retracted				:= G_IO.arDI[offsetIn+3].Ch[6];
GVL.pm[iRm*2+1].inConv.valve[2].extended				:= G_IO.arDI[offsetIn+3].Ch[7];
GVL.pm[iRm*2+1].inConv.valve[2].retracted				:= G_IO.arDI[offsetIn+3].Ch[8];
GVL.pm[iRm*2+1].outConv.photo_sensor[0]				:= G_IO.arDI[offsetIn+3].Ch[9];
GVL.pm[iRm*2+1].outConv.photo_sensor[1]				:= G_IO.arDI[offsetIn+3].Ch[10];
GVL.pm[iRm*2+1].outConv.valve[0].extended				:= G_IO.arDI[offsetIn+3].Ch[11];
GVL.pm[iRm*2+1].outConv.valve[0].retracted			:= G_IO.arDI[offsetIn+3].Ch[12];
GVL.pm[iRm*2+1].outConv.valve[1].extended				:= G_IO.arDI[offsetIn+3].Ch[13];
GVL.pm[iRm*2+1].outConv.valve[1].retracted			:= G_IO.arDI[offsetIn+3].Ch[14];
GVL.pm[iRm*2+1].inConv.photo_sensor[0]				:= G_IO.arDI[offsetIn+4].Ch[8];
GVL.pm[iRm*2+1].inConv.photo_sensor[1]				:= G_IO.arDI[offsetIn+4].Ch[9];
GVL.pm[iRm*2+1].inConv.photo_sensor[2]				:= G_IO.arDI[offsetIn+4].Ch[10];
GVL.pm[iRm*2+1].inConv.photo_sensor[3]				:= G_IO.arDI[offsetIn+4].Ch[11];
GVL.pm[iRm*2+1].inConv.photo_sensor[4]				:= G_IO.arDI[offsetIn+4].Ch[12];
GVL.pm[iRm*2+1].inConv.photo_sensor[5]				:= G_IO.arDI[offsetIn+4].Ch[13];

G_IO.arDO[offsetOut].Ch[5]	:= GVL.pm[iRm*2+1].buffer[0].power_axis;
G_IO.arDO[offsetOut].Ch[6]	:= GVL.pm[iRm*2+1].buffer[0].magnet;
G_IO.arDO[offsetOut].Ch[7]	:= GVL.pm[iRm*2+1].buffer[1].power_axis;
G_IO.arDO[offsetOut].Ch[8]	:= GVL.pm[iRm*2+1].buffer[1].magnet;
G_IO.arDO[offsetOut].Ch[9]	:= GVL.pm[iRm*2+1].power_robot;
G_IO.arDO[offsetOut].Ch[14]	:= GVL.pm[iRm*2+1].buffer[0].lamp_button;
G_IO.arDO[offsetOut].Ch[15]	:= GVL.pm[iRm*2+1].buffer[1].lamp_button;
	
G_IO.arDO[offsetOut+1].Ch[3]	:= GVL.pm[iRm*2+1].inConv.valve[0].retract;
G_IO.arDO[offsetOut+1].Ch[4]	:= GVL.pm[iRm*2+1].inConv.valve[1].retract;
G_IO.arDO[offsetOut+1].Ch[5]	:= GVL.pm[iRm*2+1].inConv.valve[2].retract;
G_IO.arDO[offsetOut+1].Ch[8]	:= GVL.pm[iRm*2+1].outConv.valve[0].retract;
G_IO.arDO[offsetOut+1].Ch[9]	:= GVL.pm[iRm*2+1].outConv.valve[1].retract;	

GVL.pm[iRm*2].contactor_inConv			:= G_IO.arDI[offsetIn+4].Ch[0];//pm[0] and pm[1]
GVL.pm[iRm*2].contactor_outConv			:= G_IO.arDI[offsetIn+4].Ch[1];//pm[0] and pm[1]
GVL.pm[iRm*2+1].contactor_inConv			:= G_IO.arDI[offsetIn+4].Ch[0];//pm[0] and pm[1]
GVL.pm[iRm*2+1].contactor_outConv			:= G_IO.arDI[offsetIn+4].Ch[1];//pm[0] and pm[1]

rTrig_power_inConv(CLK:=GVL.pm[iRm*2].power_inConv OR GVL.pm[iRm*2+1].power_inConv);
fTrig_power_inConv(CLK:=GVL.pm[iRm*2].power_inConv AND GVL.pm[iRm*2+1].power_inConv);
rTrig_power_outConv(CLK:=GVL.pm[iRm*2].power_outConv OR GVL.pm[iRm*2+1].power_outConv);
fTrig_power_outConv(CLK:=GVL.pm[iRm*2].power_outConv AND GVL.pm[iRm*2+1].power_outConv);

IF rTrig_power_inConv.Q THEN
	GVL.pm[iRm*2].power_inConv	:= TRUE;
	GVL.pm[iRm*2+1].power_inConv	:= TRUE;
END_IF
IF fTrig_power_inConv.Q THEN
	GVL.pm[iRm*2].power_inConv	:= FALSE;
	GVL.pm[iRm*2+1].power_inConv	:= FALSE;
END_IF
IF rTrig_power_outConv.Q THEN
	GVL.pm[iRm*2].power_outConv	:= TRUE;
	GVL.pm[iRm*2+1].power_outConv	:= TRUE;
END_IF
IF fTrig_power_outConv.Q THEN
	GVL.pm[iRm*2].power_outConv	:= FALSE;
	GVL.pm[iRm*2+1].power_outConv	:= FALSE;
END_IF
G_IO.arDO[offsetOut].Ch[10]	:= GVL.pm[iRm*2].power_inConv OR GVL.pm[iRm*2+1].power_inConv;//pm[0] and pm[1]
G_IO.arDO[offsetOut].Ch[11]	:= GVL.pm[iRm*2].power_outConv OR GVL.pm[iRm*2+1].power_outConv;//pm[0] and pm[1]

END_FUNCTION_BLOCK

// ---- POUs/FB_pmAxisMapping.TcPOU
FUNCTION_BLOCK FB_pmAxisMapping
VAR_INPUT
	iPM	: INT;
	iBuffer	: INT;
	sNetID	: STRING;
	nSlaveAddr : UINT;
END_VAR
VAR_OUTPUT
END_VAR
VAR
END_VAR

//========== Axis Config ==========
GVL.pm[iPM].buffer[iBuffer].mcAxis
(
	ZSN		:= TRUE,
	ZSP		:= TRUE,
	IN_OUT	:= GVL.pm[iPM].buffer[iBuffer].st_mcAxis, 
	AXIS	:= GVL.pm[iPM].buffer[iBuffer].Axisref, 
);
GVL.pm[iPM].buffer[iBuffer].st_mcAxis.bPosSensorShow	:= FALSE;
GVL.pm[iPM].buffer[iBuffer].st_mcAxis.bNegSensorShow	:= FALSE;
GVL.pm[iPM].buffer[iBuffer].st_mcAxis.bStopButtonShow	:= TRUE;
GVL.pm[iPM].buffer[iBuffer].st_mcAxis.rMaxAcceleration	:= 50000;
GVL.pm[iPM].buffer[iBuffer].st_mcAxis.rMaxDeceleration	:= 50000;
GVL.pm[iPM].buffer[iBuffer].st_mcAxis.rMaxJerk			:= 500000;
GVL.pm[iPM].buffer[iBuffer].st_mcAxis.rAcceleration	:= 2500;
GVL.pm[iPM].buffer[iBuffer].st_mcAxis.rDeceleration	:= 2500;
GVL.pm[iPM].buffer[iBuffer].st_mcAxis.rJerk			:= 12500;
GVL.pm[iPM].buffer[iBuffer].st_mcAxis.rMaxVelocity		:= 100;
GVL.pm[iPM].buffer[iBuffer].st_mcAxis.rMaxDistance		:= 50;
GVL.pm[iPM].buffer[iBuffer].st_mcAxis.bPosSen	:= TRUE ;
GVL.pm[iPM].buffer[iBuffer].st_mcAxis.bNegSen	:= TRUE ;
GVL.pm[iPM].buffer[iBuffer].st_mcAxis.mcHome.bCalibrationCam	:= GVL.pm[iPM].buffer[iBuffer].axis_sensor;
GVL.pm[iPM].buffer[iBuffer].st_mcAxis.bPositionSensor	:= GVL.pm[iPM].buffer[iBuffer].axis_sensor;
GVL.pm[iPM].buffer[iBuffer].st_mcAxis.bdirFW	:= TRUE;
GVL.pm[iPM].buffer[iBuffer].st_mcAxis.rSetPos	:= 0;
GVL.pm[iPM].buffer[iBuffer].st_mcAxis.sNetID := sNetID;
GVL.pm[iPM].buffer[iBuffer].st_mcAxis.nSlaveAddr	:= nSlaveAddr;

END_FUNCTION_BLOCK

// ---- POUs/FB_axisCtrl.TcPOU
FUNCTION_BLOCK FB_axisCtrl
VAR_INPUT
	
END_VAR
VAR_OUTPUT
END_VAR
VAR_IN_OUT     
	stAxisCtrl	:ST_axisCtrl; 	
	IN_OUT 		: ST_MotionAxis_MC	;//struct for each axis
END_VAR
VAR
	ton_delay	: TON;
END_VAR

//add timeout for this fuction block
ton_delay(PT:= T#2S);
CASE stAxisCtrl.iCmd OF
	0:
		IN_OUT.mcReset.Execute	:= FALSE;
		IN_OUT.mcStop.Execute	:= FALSE	;
	1:
		IN_OUT.mcPower.Enable	:= TRUE;
		stAxisCtrl.iCmd	:= 0;
	2:
		IN_OUT.mcPower.Enable	:= FALSE;
		stAxisCtrl.iCmd	:= 0;	
	3:
		IN_OUT.mcReset.Execute	:= TRUE;
		stAxisCtrl.iCmd	:= 0;
	4:
		IN_OUT.mcStop.Execute	:= TRUE;
		stAxisCtrl.iCmd	:= 0;	
	5: 
		IN_OUT.mcMoveAbsolute.Execute := TRUE;
		IN_OUT.rActualPosSet	:= stAxisCtrl.rPosition;
		IN_OUT.rVelocitySet	:= stAxisCtrl.iSpeed;
		IF IN_OUT.mcMoveAbsolute.Done THEN
			stAxisCtrl.iCmd	:= 0;
		END_IF
		
	10://REM aging test start
		ton_delay.IN	:= FALSE;
		IN_OUT.mcMoveAbsolute.Execute := TRUE;
		IN_OUT.rActualPosSet	:= 0;
		IN_OUT.rVelocitySet	:= stAxisCtrl.iSpeed;
		IF IN_OUT.mcMoveAbsolute.Done THEN
			IN_OUT.mcMoveAbsolute.Execute := FALSE;
			stAxisCtrl.iCmd	:= 11;
		END_IF
	11:
		ton_delay.IN	:= TRUE;
		IF ton_delay.Q THEN
			stAxisCtrl.iCmd	:= 12;
		END_IF
	12:
		ton_delay.IN	:= FALSE;
		IN_OUT.mcMoveAbsolute.Execute := TRUE;
		IN_OUT.rActualPosSet	:= stAxisCtrl.rPosition;
		IN_OUT.rVelocitySet	:= stAxisCtrl.iSpeed;
		IF IN_OUT.mcMoveAbsolute.Done THEN
			IN_OUT.mcMoveAbsolute.Execute := FALSE;
			stAxisCtrl.iCmd	:= 13;
		END_IF
	13:
		ton_delay.IN	:= TRUE;
		IF ton_delay.Q THEN
			stAxisCtrl.iCmd	:= 10;
		END_IF	
	
		
	20://PM buffer aging test start
		ton_delay.IN	:= FALSE;
		IN_OUT.mcMoveRelative.Execute := TRUE;
		IN_OUT.rPosition	:= stAxisCtrl.rPosition;
		IN_OUT.rVelocity	:= stAxisCtrl.iSpeed;
		IF IN_OUT.mcMoveRelative.Done THEN
			IN_OUT.mcMoveRelative.Execute := FALSE;
			stAxisCtrl.iCmd	:= 21;
		END_IF
	21:
		ton_delay.IN	:= TRUE;
		IF ton_delay.Q THEN
			stAxisCtrl.iCmd	:= 20;
		END_IF


	
	100:
		IN_OUT.mcMoveAbsolute.Execute := FALSE;
		IN_OUT.mcMoveVelocity.Execute	:= FALSE;
		IN_OUT.mcMoveRelative.Execute	:= FALSE;
		IN_OUT.mcStop.Execute	:= TRUE;
		stAxisCtrl.iCmd	:= 0;
		
END_CASE;
stAxisCtrl.iStatus := stAxisCtrl.iCmd;

END_FUNCTION_BLOCK

// ---- GVLs/kitting deca/FB_Converter.TcPOU
FUNCTION_BLOCK FB_Converter 
VAR_INPUT
	
	iMotor	: WORD;
	bSetParaEx	: BOOL;
	cmd  AT%Q*	: UINT;
	freq AT%Q*	: UINT;

	reset	: BOOL;
END_VAR
VAR_OUTPUT
	status	AT%I*	:  UINT;//Bit0：运行状态；Bit1：正反转状态；Bit2：是否发生故障
							//Bit3：输出频率是否到达设定频率；Bit4：通信正常标志；
							//Bit5~Bit7：保留；Bit8~Bit15：故障主码
	running_freq	AT%I*	:  UINT;
	xErr	:  BOOL;
	errorID	: UINT;
	xDone	: BOOL;
END_VAR
VAR_IN_OUT
	stConverter	: ST_Converter;
	//sNetID : STRING;
	//nSlaveAddr	:UINT;
	
END_VAR
VAR
	iCase	: INT;
	i : INT;
	coeWrt		:	FB_EcCoESdoWrite;
	coeRead		:  	FB_EcCoESdoRead;
	nSubIndex	: BYTE;
	nIndex		: WORD;
	iSdoWrite	: INT; 
	iSdoRead	: INT;
	offset: WORD;
	rtrig_bSetPara	: R_TRIG;
	rtrig_bReset	: R_TRIG;
	ton_delay	: TON;
END_VAR

xDone	:= FALSE; 
coeWrt(
	sNetId:= stConverter.sNetID, 
	nSlaveAddr:=stConverter.nSlaveAddr, 
	nSubIndex:= nSubIndex, 
	nIndex:= nIndex, 
	pSrcBuf:= ADR(iSdoWrite), 
	cbBufLen:= SIZEOF(iSdoWrite), 
	bExecute:= , 
	tTimeout:= , 
	bBusy=> , 
	bError=> , 
	nErrId=> );
coeRead(
	sNetId:= stConverter.sNetID, 
	nSlaveAddr:=stConverter.nSlaveAddr, 
	nSubIndex:= nSubIndex, 
	nIndex:= nIndex, 
	pDstBuf:= ADR(iSdoRead), 
	cbBufLen:= SIZEOF(iSdoRead), 
	bExecute:= , 
	tTimeout:= , 
	bBusy=> , 
	bError=> , 
	nErrId=> );

(*
addr		valve					comment	
整流单元								
FD-10		3					通信协议选择(面板设定)	
逆变单元								
F0:02		2					control mode	
F0:03		2					command source selection	
F0:04		9					main frequency source X selection	
F0:0B		6000					maximum frequency	
F0:0D		6000					frequency upper limit	
F0:12		5					acceleration time 1	
F0:13		5					deceleration time 1	
F0:14		1					acceleration/deceleration time unit	
F1:01		1					motor type	
F1:02		1					rated motor power	
F1:03		220					rated motor voltage	
F1:04		6					rated motor current	
F1:05		6000					rated motor frequency	
F1:06		1600					rated motor speed	
*)

offset	:= 16#800*iMotor;
//control mode
stConverter.nIndex[0]	:= 16#20F0+offset;
stConverter.nSubIndex[0]	:= 16#02;
stConverter.iSdoWrite[0]	:= 2;
//command source selection
stConverter.nIndex[1]	:= 16#20F0+offset;
stConverter.nSubIndex[1]	:= 16#03;
stConverter.iSdoWrite[1]	:= 2;
//main frequency source X selection
stConverter.nIndex[2]	:= 16#20F0+offset;
stConverter.nSubIndex[2]	:= 16#04;
stConverter.iSdoWrite[2]	:= 9;
//maximum frequency
stConverter.nIndex[3]	:= 16#20F0+offset;
stConverter.nSubIndex[3]	:= 16#0B;
stConverter.iSdoWrite[3]	:= 6000;
//frequency upper limit
stConverter.nIndex[4]	:= 16#20F0+offset;
stConverter.nSubIndex[4]	:= 16#0D;
stConverter.iSdoWrite[4]	:= 6000;
//acceleration time 1
stConverter.nIndex[5]	:= 16#20F0+offset;
stConverter.nSubIndex[5]	:= 16#12;
stConverter.iSdoWrite[5]	:= 5;
//deceleration time 1
stConverter.nIndex[6]	:= 16#20F0+offset;
stConverter.nSubIndex[6]	:= 16#13;
stConverter.iSdoWrite[6]	:= 5;
//acceleration/deceleration time unit	
stConverter.nIndex[7]	:= 16#20F0+offset;
stConverter.nSubIndex[7]	:= 16#14;
stConverter.iSdoWrite[7]	:= 1;
//motor type	
stConverter.nIndex[8]	:= 16#20F1+offset;
stConverter.nSubIndex[8]	:= 16#01;
stConverter.iSdoWrite[8]	:= 1;
//rated motor power	
stConverter.nIndex[9]	:= 16#20F1+offset;
stConverter.nSubIndex[9]	:= 16#02;
stConverter.iSdoWrite[9]	:= 1;
//rated motor voltage		
stConverter.nIndex[10]	:= 16#20F1+offset;
stConverter.nSubIndex[10]	:= 16#03;
stConverter.iSdoWrite[10]	:= 220;
//rated motor current		
stConverter.nIndex[11]	:= 16#20F1+offset;
stConverter.nSubIndex[11]	:= 16#04;
stConverter.iSdoWrite[11]	:= 6;
//rated motor frequency		
stConverter.nIndex[12]	:= 16#20F1+offset;
stConverter.nSubIndex[12]	:= 16#05;
stConverter.iSdoWrite[12]	:= 6000;
//rated motor speed		
stConverter.nIndex[13]	:= 16#20F1+offset;
stConverter.nSubIndex[13]	:= 16#06;
stConverter.iSdoWrite[13]	:= 1600;

ton_delay(PT:= T#0.1S);
rtrig_bSetPara(CLK:=bSetParaEx);
rtrig_bReset(CLK:=reset);
CASE iCase OF
	0:
		coeWrt.bExecute	:= FALSE;
		ton_delay.IN	:= FALSE;
		i:=0;
		xDone	:= FALSE;
		IF rtrig_bSetPara.Q THEN
			iCase	:= 1;
		END_IF	
		IF rtrig_bReset.Q THEN
			iCase	:= 10;
		END_IF				
	1: 
		nIndex	:= stConverter.nIndex[i];
		nSubIndex	:= stConverter.nSubIndex[i];
		iSdoWrite	:= stConverter.iSdoWrite[i];
		i	:= i+1;
		coeWrt.bExecute	:= TRUE;
		iCase	:= 2;
	2:
		ton_delay.IN	:= TRUE;
		IF ton_delay.Q THEN
			iCase	:= 3;
		END_IF		
	3:
		ton_delay.IN	:= FALSE;
		coeWrt.bExecute	:= FALSE;
		IF i >13 THEN
			iCase	:= 0;
			xDone	:= TRUE;
			//RETURN ;
		ELSE
			iCase	:= 1;
		END_IF	
	10: 
		IF status.2 THEN
			cmd	:=INT_TO_UINT(E_CMD_ConverterMotor.RESET);
		END_IF
		iCase	:= 11;
	11:
		ton_delay.IN	:= TRUE;
		IF ton_delay.Q THEN
			iCase	:= 0;
		END_IF		
END_CASE


xErr	:= status.2 ;

errorID	:= SHR(status,8);

METHOD M_SetPara : BOOL
VAR_INPUT
	//iMotor	: WORD;
	
END_VAR
VAR_IN_OUT
	
END_VAR
VAR

END_VAR

(*FOR i:=0 TO 13 DO
	nIndex	:= stConverter.nIndex[i];
	nSubIndex	:= stConverter.nSubIndex[i];
	iSdoWrite	:= stConverter.iSdoWrite[i];
	CoeWrt.bExecute	:= TRUE;
END_FOR*)
END_METHOD

END_FUNCTION_BLOCK

// ---- POUs/FB_lcIOmapping.TcPOU
FUNCTION_BLOCK FB_lcIOmapping
VAR_INPUT
	iLc	: INT;
	mcAxis	: FB_MotionAxis_MC;	
	sNetID	: STRING;
	nSlaveAddr : UINT;
END_VAR
VAR_OUTPUT
END_VAR
VAR_IN_OUT
	IN_OUT	: ST_MotionAxis_MC;
END_VAR
VAR
	offset	: INT;
END_VAR

offset:= 85+iLc*3;
GVL.lc[iLc].rollerIn.roller.err					:= G_IO.arDI[offset].Ch[0];
GVL.lc[iLc].rollerIn.photo_sensor				:= G_IO.arDI[offset].Ch[1];
GVL.lc[iLc].rollerOut.roller.err				:= G_IO.arDI[offset].Ch[2];
GVL.lc[iLc].rollerOut.photo_sensor				:= G_IO.arDI[offset].Ch[3];
GVL.lc[iLc].contactor_beltConv					:= G_IO.arDI[offset].Ch[4];
GVL.lc[iLc].belt_out.photo_sensor[0]			:= G_IO.arDI[offset].Ch[5];
GVL.lc[iLc].belt_out.photo_sensor[1]			:= G_IO.arDI[offset].Ch[6];
GVL.lc[iLc].belt_out.photo_sensor[2]			:= G_IO.arDI[offset].Ch[7];
GVL.lc[iLc].lateral.contactor_axis				:= G_IO.arDI[offset].Ch[8];
GVL.lc[iLc].lateral.limit_sensor[0]				:= G_IO.arDI[offset].Ch[9];
GVL.lc[iLc].lateral.limit_sensor[1]				:= G_IO.arDI[offset].Ch[10];
GVL.lc[iLc].lateral.limit_sensor[2]				:= G_IO.arDI[offset].Ch[11];
GVL.lc[iLc].lateral.valve_lift.extended			:= G_IO.arDI[offset].Ch[12];
GVL.lc[iLc].lateral.valve_lift.retracted		:= G_IO.arDI[offset].Ch[13];
GVL.lc[iLc].lateral.valve_clamp[0].extended			:= G_IO.arDI[offset].Ch[14];
GVL.lc[iLc].lateral.valve_clamp[0].retracted		:= G_IO.arDI[offset].Ch[15];
GVL.lc[iLc].lateral.valve_clamp[1].extended			:= G_IO.arDI[offset+1].Ch[0];
GVL.lc[iLc].lateral.valve_clamp[1].retracted		:= G_IO.arDI[offset+1].Ch[1];
GVL.lc[iLc].valve_stopper[0].extended			:= G_IO.arDI[offset+1].Ch[2];
GVL.lc[iLc].valve_stopper[0].retracted			:= G_IO.arDI[offset+1].Ch[3];
GVL.lc[iLc].valve_stopper[1].extended			:= G_IO.arDI[offset+1].Ch[4];
GVL.lc[iLc].valve_stopper[1].retracted			:= G_IO.arDI[offset+1].Ch[5];
GVL.lc[iLc].valve_guide[0].extended				:= G_IO.arDI[offset+1].Ch[6];
GVL.lc[iLc].valve_guide[0].retracted			:= G_IO.arDI[offset+1].Ch[7];
GVL.lc[iLc].valve_guide[1].extended				:= G_IO.arDI[offset+1].Ch[8];
GVL.lc[iLc].valve_guide[1].retracted			:= G_IO.arDI[offset+1].Ch[9];
GVL.lc[iLc].pressure_sensor						:= G_IO.arDI[offset+1].Ch[10];

G_IO.arDO[offset].Ch[0]		:= GVL.lc[iLc].rollerIn.roller.Power;
G_IO.arDO[offset].Ch[1]		:= GVL.lc[iLc].rollerIn.roller.forward;
G_IO.arDO[offset].Ch[2]		:= GVL.lc[iLc].rollerIn.roller.backward;
G_IO.arDO[offset].Ch[3]		:= GVL.lc[iLc].rollerOut.roller.Power;
G_IO.arDO[offset].Ch[4]		:= GVL.lc[iLc].rollerOut.roller.forward;
G_IO.arDO[offset].Ch[5]		:= GVL.lc[iLc].rollerOut.roller.backward;
G_IO.arDO[offset].Ch[6]		:= GVL.lc[iLc].power_beltConv;
G_IO.arDO[offset].Ch[7]		:= GVL.lc[iLc].lateral.power_axis;
G_IO.arDO[offset].Ch[8]		:= GVL.lc[iLc].lateral.valve_lift.extend;
G_IO.arDO[offset].Ch[9]		:= GVL.lc[iLc].lateral.valve_lift.retract;
G_IO.arDO[offset].Ch[10]	:= GVL.lc[iLc].lateral.valve_clamp[0].retract;
G_IO.arDO[offset].Ch[11]	:= GVL.lc[iLc].lateral.valve_clamp[1].retract;
G_IO.arDO[offset].Ch[12]	:= GVL.lc[iLc].valve_stopper[0].retract;
G_IO.arDO[offset].Ch[13]	:= GVL.lc[iLc].valve_stopper[1].retract;
G_IO.arDO[offset].Ch[14]	:= GVL.lc[iLc].valve_guide[0].extend;
G_IO.arDO[offset].Ch[15]	:= GVL.lc[iLc].valve_guide[1].extend;


mcAxis(
	ZSN		:= GVL.lc[iLc].lateral.limit_sensor[2]	 OR IN_OUT.xHoming,
	ZSP		:= GVL.lc[iLc].lateral.limit_sensor[1]		OR IN_OUT.xHoming,
	IN_OUT	:= IN_OUT, 
	AXIS	:= GVL.lc[iLc].lateral.AxisRef, 
);
IN_OUT.bPosSensorShow	:= TRUE;
IN_OUT.bNegSensorShow	:= TRUE;
IN_OUT.bStopButtonShow	:= TRUE;
IN_OUT.rMaxAcceleration	:= 50000;
IN_OUT.rMaxDeceleration	:= 50000;
IN_OUT.rMaxJerk			:= 500000;
IN_OUT.rAcceleration	:= 2500;
IN_OUT.rDeceleration	:= 2500;
IN_OUT.rJerk			:= 12500;
IN_OUT.rMaxVelocity		:= 100;
IN_OUT.rMaxDistance		:= 50;
IN_OUT.bPosSen	:= GVL.lc[iLc].lateral.limit_sensor[1] ;
IN_OUT.bNegSen	:= GVL.lc[iLc].lateral.limit_sensor[2] ;
IN_OUT.mcHome.bCalibrationCam	:= GVL.lc[iLc].lateral.limit_sensor[0];
IN_OUT.bPositionSensor	:= GVL.lc[iLc].lateral.limit_sensor[0];
IN_OUT.bdirFW	:= TRUE;
IN_OUT.rSetPos	:= 0;
IN_OUT.sNetID := sNetID;
IN_OUT.nSlaveAddr	:= nSlaveAddr;

END_FUNCTION_BLOCK

// ---- GVLs/kitting deca/axis/FB_MotionAxis_MC.TcPOU
FUNCTION_BLOCK FB_MotionAxis_MC

VAR_INPUT
	ZSN	   			: BOOL												;
	ZSP				: BOOL												; 
	Exceeding_us			: INT;
	sNameAxis				: STRING [40];

END_VAR         	
                	
VAR  
	rtFirstCycle	: R_TRIG;						
	mcHomeAxis		: 	MC_HomeAxis						;//ADD BY EVAN 
	sAxisName		: STRING											;//Axis name          	
	xPlus			: BOOL												;	
	xMinus			: BOOL												;
	bDone			: BOOL												;	

// Variables for Hard Stop Homing	                        			
	iStatehsHomig	: E_HomingSteps := E_HomingSteps.IDLE				;
	rtHome			: R_TRIG											;
	rtHomeReset		: R_TRIG											;
	tonTimeOut		: TON												;
	xTimerStart		: BOOL												;
	bLSDefaultVal	: BOOL												; // Save Def value from driver
	xHomeError		: BOOL												;
// Variables for Force Control          					

	rtForceC		: R_TRIG											;
	rtForceCReset	: R_TRIG											;
	DelMaxPos		: LREAL 											;
	rCurrLimit		: LREAL												;
	StartPos		: LREAL												;
	xForceCError	: BOOL												;
//	Variables for Backlash Compensation
	rLastMove		: LREAL := 1										;
	tonBackComp		: TON												;
	rBacklashPer	: LREAL												;	
	
// Variables for errors
	rtError					:	R_TRIG;
	pTextType				:	POINTER TO STRING;
	sAxisErrorID			:	STRING(10);	
	ErrorMSG				:	STRING[255];

//	Exceeding time measuring
	sysTime					:	GETCPUCOUNTER;//GETSYSTEMTIME;					//	Used to measure execution time.
	uStartTime				:	UDINT;
	uFinishTime				:	UDINT;
	ftimeDiff				:	REAL;
	ton_dly	: TON;
END_VAR         	
                	
VAR_IN_OUT      	
	IN_OUT 			: ST_MotionAxis_MC	;//struct for each axis
	AXIS 			: AXIS_REF			;//Axis obj	
END_VAR

VAR_OUTPUT
	xError			: BOOL				;
	xBusy			: BOOL				;
END_VAR
VAR CONSTANT
	parallelGroupTLName		:	STRING := 'Port_851.TL_Axis_Error';
END_VAR

(* Power options ********************************************************************************************)			
IN_OUT.mcPower(
	Axis				:= AXIS, 
	Enable				:= , 
	Enable_Positive		:= ZSP, 
	Enable_Negative		:= ZSN OR IN_OUT.mcHome.Busy, 
	Override			:= , 
	BufferMode			:= , 
	Options				:= , 
	Status				=> , 
	Busy				=> , 
	Active				=> , 
	Error				=> , 
	ErrorID				=> );
	
(* Halt Mode ********************************************************************************************)	
IN_OUT.mcHalt(
	Axis				:= AXIS, 
	Execute				:= , 
	Deceleration		:= IN_OUT.rDeceleration, 
	Jerk				:= , 
	BufferMode			:= , 
	Options				:= , 
	Done				=> , 
	Busy				=> , 
	Active				=> , 
	CommandAborted		=> , 
	Error				=> , 
	ErrorID				=> );
	
(* Homing ***********************************************************************************************)
IN_OUT.mcHome(
	Axis				:= AXIS, 
	Execute				:= , 
	Position			:= in_out.rFirstpos, 
	HomingMode			:= MC_Direct, 
	BufferMode			:= , 
	Options				:= , 
	bCalibrationCam		:= ,//NOT  ZSN, 
	Done				=> , 
	Busy				=> , 
	Active				=> , 
	CommandAborted		=> , 
	Error				=> , 
	ErrorID				=> );
	
(* JOG **************************************************************************************************)
IN_OUT.mcJog(
	Axis				:= AXIS, 
	JogForward			:= , 
	JogBackwards		:= , 
	Mode				:= E_JogMode.MC_JOGMODE_CONTINOUS, 
	Position			:= , 
	Velocity			:= IN_OUT.rVelocity, 
	Acceleration		:= IN_OUT.rAcceleration, 
	Deceleration		:= IN_OUT.rDeceleration, 
	Jerk				:= IN_OUT.rJerk, 
	Done				=> , 
	Busy				=> , 
	Active				=> , 
	CommandAborted		=> , 
	Error				=> , 
	ErrorID				=> );
	
(* Move Absolute ****************************************************************************************)	
IN_OUT.mcMoveAbsolute(
	Axis				:= AXIS, 
	Execute				:= , 
	Position			:= IN_OUT.rActualPosSet, 
	Velocity			:= IN_OUT.rVelocitySet,     
	Acceleration		:= IN_OUT.rAcceleration, 
	Deceleration		:= IN_OUT.rDeceleration, 
	Jerk				:= IN_OUT.rJerk,         
	BufferMode			:= , 
	Options				:= , 
	Done				=> , 
	Busy				=> , 
	Active				=> , 
	CommandAborted		=> , 
	Error				=> , 
	ErrorID				=> );

	IF IN_OUT.bMoveAbsHMI THEN
		IN_OUT.mcMoveAbsolute.Execute	:= TRUE;
		IN_OUT.rActualPosSet	:= IN_OUT.rActualPosHMI;
		IN_OUT.rVelocitySet		:= IN_OUT.rVeloPers;
	END_IF
(* Move Relative *********************************************************************************************************)
IN_OUT.mcMoveRelative(
	Axis				:= AXIS, 
	Execute				:= , 
	Distance			:= IN_OUT.rPosition + IN_OUT.rBacklashvalue, 
	Velocity			:= IN_OUT.rVelocity,      
	Acceleration		:= IN_OUT.rAcceleration,  
	Deceleration		:= IN_OUT.rDeceleration,  
	Jerk				:= IN_OUT.rJerk,          
	BufferMode			:= ,
	Options				:= , 
	Done				=> bDone, 
	Busy				=> , 
	Active				=> , 
	CommandAborted		=> , 
	Error				=> , 
	ErrorID				=> );
	
(* Move Velocity *********************************************************************************************************)
	
IN_OUT.mcMoveVelocity(
	Axis				:=	AXIS,
	Execute				:=	,
	Velocity			:=	IN_OUT.rVelocity,
	Acceleration		:=	IN_OUT.rAcceleration,
	Deceleration		:=	IN_OUT.rDeceleration,
	Jerk				:=	IN_OUT.rJerk,
	Direction			:=	IN_OUT.axisDirection,
	BufferMode			:=	,
	Options				:=	,
	InVelocity			=>	,
	Busy				=>	,
	Active				=>	,
	CommandAborted		=>	,
	Error				=>	,
	ErrorID				=>	);
	
(**)	
IN_OUT.mcReadStatus(
	Axis				:= AXIS, 
	Enable				:= TRUE, 
	Valid				=> , 
	Busy				=> , 
	Error				=> , 
	ErrorID				=> , 
	ErrorStop			=> , 
	Disabled			=> , 
	Stopping			=> , 
	StandStill			=> , 
	DiscreteMotion		=> , 
	ContinuousMotion	=> , 
	SynchronizedMotion	=> , 
	Homing				=> , 
	ConstantVelocity	=> , 
	Accelerating		=> , 
	Decelerating		=> , 
	Status				=> );
	
(* Reset ************************************************************************************************)
IN_OUT.mcReset(
	Axis				:= AXIS, 
	Execute				:= , 
	Done				=> , 
	Busy				=> , 
	Error				=> , 
	ErrorID				=> );
	
(* Stop *************************************************************************************************)
IN_OUT.mcStop(
	Axis				:= AXIS, 
	Execute				:= , 
	Deceleration		:= , 
	Jerk				:= , 
	Options				:= , 
	Done				=> , 
	Busy				=> , 
	Active				=> , 
	CommandAborted		=> , 
	Error				=> , 
	ErrorID				=> );

(* Set Position *************************************************************************************************)
in_out.mcSetpoint(
	Axis			 := AXIS, 
	Execute			 := , 
	Position		 := IN_OUT.rSetPos, 
	Mode			 := , 
	Options			 := , 
	Done			 => , 
	Busy			 => , 
	Error			 => , 
	ErrorID			 => );


(* write status *************************************************************************************************)
IN_OUT.mcWriteBoolParameter(
	Axis			:= 	AXIS, 
	Execute:= 				, 
	ParameterNumber:= 		, 
	Value:= , 
	Done=> , 
	Busy=> , 
	Error=> , 
	ErrorID=> );

(* Read status *************************************************************************************************)
IN_OUT.mcReadBoolParameter(
	Axis:= AXIS, 
	Enable:= , 
	ParameterNumber:= , 
	ReadMode:= , 
	Valid=> , 
	Busy=> , 
	Error=> , 
	ErrorID=> , 
	Value=> );	

(*Read Actualposition***************************************************************)
IN_OUT.mcReadActualPosition(
	Axis:= AXIS, 
	Enable:= TRUE, 
	Valid=> , 
	Busy=> , 
	Error=> , 
	ErrorID=> , 
	Position=> IN_OUT.rActualPos );   
(*COE write**************************************************************************)	

IN_OUT.CoeWrt(
	sNetId:= IN_OUT.sNetID, 
	nSlaveAddr:= IN_OUT.nSlaveAddr, 
	nSubIndex:= IN_OUT.nSubIndex, 
	nIndex:= IN_OUT.nIndex, 
	pSrcBuf:= ADR(IN_OUT.iSdoWrite), 
	cbBufLen:= SIZEOF(IN_OUT.iSdoWrite), 
	bExecute:= , 
	tTimeout:= , 
	bBusy=> , 
	bError=> , 
	nErrId=> );
	ton_dly(PT:=T#100MS);
CASE IN_OUT.iCoeWrt OF 
	0:
		IN_OUT.CoeWrt.bExecute := FALSE;
	1:
		IN_OUT.CoeWrt.bExecute := TRUE;
		IN_OUT.nIndex	:= 16#2005;
		IN_OUT.nSubIndex	:= 16#1F;
		IN_OUT.iSdoWrite	:= 6;//clear encoder and set current position as origin
		IN_OUT.iCoeWrt	:= 10;
	2:
		IN_OUT.CoeWrt.bExecute := TRUE;
		IN_OUT.nIndex	:= 16#2002;
		IN_OUT.nSubIndex	:= 16#02;
		IN_OUT.iSdoWrite	:= 1;//linear mode
		IN_OUT.iCoeWrt	:= 10;
	3:
		IN_OUT.CoeWrt.bExecute := TRUE;
		IN_OUT.nIndex	:= 16#2002;
		IN_OUT.nSubIndex	:= 16#02;
		IN_OUT.iSdoWrite	:= 2;//rotate mode
		IN_OUT.iCoeWrt	:= 10;
	4:
		IN_OUT.CoeWrt.bExecute := TRUE;
		IN_OUT.nIndex	:= 16#2004;
		IN_OUT.nSubIndex	:= 16#06;
		IN_OUT.iSdoWrite	:= 1;//breaker on
		IN_OUT.iCoeWrt	:= 10;
	5:
		IN_OUT.CoeWrt.bExecute := TRUE;
		IN_OUT.nIndex	:= 16#2004;
		IN_OUT.nSubIndex	:= 16#06;
		IN_OUT.iSdoWrite	:= 0;//breaker off
		IN_OUT.iCoeWrt	:= 10;		
	10:		
		IN_OUT.iCoeWrt	:= 0;
END_CASE







	(*mcHomeAxis***************************************************************)
	mcHomeAxis(
		xExecute:= , 
		xReset:= , 
		InOut:=IN_OUT , 
		xRedy=> , 
		xBusy=> , 
		xDone=> , 
		xError=> ); 
	                                                                                                              	
(******************************************************************************************************************)
	
(**error flag**)

	IN_OUT.xTorqueErr	:=ABS(IN_OUT.rActTorque)>IN_OUT.rToqueLimitSet ;

	
	

	xError := IN_OUT.mcReadStatus.Error OR xHomeError OR IN_OUT.mcMoveAbsolute.Error OR IN_OUT.xTorqueErr ;	
	rtError(CLK:= (IN_OUT.mcReadStatus.ErrorID <> 0 OR xError) AND NOT IN_OUT.xMuteAxisErrorMessages);
	
(*************************** READ ERROR FROM DRIVE *************************)
rtFirstCycle(CLK:= TRUE);
sysTime(cpuCntLoDW => uStartTime);	
sysTime(cpuCntLoDW => uFinishTime);
//M_CheckExceedingTime();

(*************************** GET AXIS ERROR MESSAGE *************************)	
	
	IF rtError.Q THEN
		IF IN_OUT.xTorqueErr THEN
			sAxisErrorID	:= 'TORQUE';
		ELSE
			sAxisErrorID	:=	TO_STRING(IN_OUT.mcReadStatus.ErrorID);
		END_IF
		IN_OUT.mcStop.Execute	:= TRUE;
	
	END_IF
(**remember the Velocity**) 
	IF IN_OUT.rVeloPers <> 0 THEN 
		IN_OUT.rVelocity:= IN_OUT.rVeloPers;
	ELSE 
		IN_OUT.rVeloPers := IN_OUT.rVelocity;	
	END_IF	
(**remember the Acceleration**)
	IF IN_OUT.rAccPers <> 0 THEN 
		IN_OUT.rAcceleration:= IN_OUT.rAccPers;
	ELSE 
		IN_OUT.rAccPers := IN_OUT.rAcceleration;		
	END_IF	
(**remember the Deceleration**)
	IF IN_OUT.rDecPers <> 0 THEN 
		IN_OUT.rDeceleration:= IN_OUT.rDecPers;
	ELSE 
		IN_OUT.rDecPers := IN_OUT.rDeceleration;		
	END_IF
(**False all Executions if function done or error**)
	IF IN_OUT.mcMoveRelative.Done OR IN_OUT.mcMoveRelative.Error OR IN_OUT.mcReset.Busy THEN 
		IN_OUT.mcMoveRelative.Execute := FALSE;
	END_IF

	IF IN_OUT.mcMoveVelocity.Error OR IN_OUT.mcReset.Busy OR IN_OUT.mcMoveVelocity.Busy THEN 
		IN_OUT.mcMoveVelocity.Execute := FALSE;
	END_IF
	
	IF IN_OUT.mcSetpoint.done OR IN_OUT.mcSetpoint.Error THEN
		IN_OUT.mcSetpoint.Execute := FALSE;
	END_IF
	
    IF  IN_OUT.mcMoveAbsolute.Done OR IN_OUT.mcMoveAbsolute.Error OR IN_OUT.mcReset.Busy THEN 
		IN_OUT.mcMoveAbsolute.Execute := FALSE;
	END_IF
 
	 IF IN_OUT.mcHome.Done OR IN_OUT.mcHome.Error THEN 
		IN_OUT.mcHome.Execute := FALSE;
	END_IF
	
	IF IN_OUT.mcStop.Done OR IN_OUT.mcStop.Error THEN 
		IN_OUT.mcStop.Execute := FALSE;
	END_IF
	
	IF IN_OUT.mcReset.Done OR IN_OUT.mcReset.Error THEN 
		IN_OUT.mcReset.Execute := FALSE;
	END_IF
			
	IF IN_OUT.mcReadBoolParameter.Valid OR IN_OUT.mcReadBoolParameter.Error THEN 
		IN_OUT.mcReadBoolParameter.Enable := FALSE;
	END_IF	
	
	IF IN_OUT.mcWriteBoolParameter.Done OR IN_OUT.mcWriteBoolParameter.Error THEN 
		IN_OUT.mcWriteBoolParameter.Execute	:= FALSE;
	END_IF	
		

	
	
	
(**Save done state into temp variable**)	
	
	IF IN_OUT.mcMoveAbsolute.Done THEN
		IN_OUT.xMoveABSDone := TRUE;
	END_IF	
	
	IF IN_OUT.mcMoveRelative.Done THEN
		IN_OUT.xMoveRelDone := TRUE;
	END_IF

PROPERTY P_AxisName : STRING
SET
sAxisName := P_AxisName;
END_SET
END_PROPERTY

PROPERTY P_CurrLimit : LREAL
SET
rCurrLimit := P_CurrLimit;
END_SET
END_PROPERTY

PROPERTY P_DelMaxPos : LREAL
SET
DelMaxPos := P_DelMaxPos;
END_SET
END_PROPERTY

PROPERTY P_ForceCError : BOOL
GET
P_ForceCError := xForceCError;
END_GET
END_PROPERTY

PROPERTY P_hsHomingError : BOOL
GET
P_hsHomingError := xHomeError;
END_GET
END_PROPERTY

PROPERTY P_StartPos : LREAL
SET
StartPos := P_StartPos;
END_SET
END_PROPERTY

END_FUNCTION_BLOCK

// ---- POUs/FB_lbIOmapping.TcPOU
FUNCTION_BLOCK FB_lbIOmapping
VAR_INPUT
	iLb	: INT;
	//sNetID	: STRING;
	//nSlaveAddr : UINT;
END_VAR
VAR_OUTPUT
END_VAR
VAR_IN_OUT
	
END_VAR
VAR
	offset	: INT;
END_VAR

offset:= 87+iLb*3;
GVL.lb[iLb].contactor_beltConv					:= G_IO.arDI[offset].Ch[0];
GVL.lb[iLb].valve_stopper[0].extended			:= G_IO.arDI[offset].Ch[1];
GVL.lb[iLb].valve_stopper[0].retracted			:= G_IO.arDI[offset].Ch[2];
GVL.lb[iLb].valve_stopper[1].extended			:= G_IO.arDI[offset].Ch[3];
GVL.lb[iLb].valve_stopper[1].retracted			:= G_IO.arDI[offset].Ch[4];
GVL.lb[iLb].valve_stopper[2].extended			:= G_IO.arDI[offset].Ch[5];
GVL.lb[iLb].valve_stopper[2].retracted			:= G_IO.arDI[offset].Ch[6];
GVL.lb[iLb].valve_stopper[3].extended			:= G_IO.arDI[offset].Ch[7];
GVL.lb[iLb].valve_stopper[3].retracted			:= G_IO.arDI[offset].Ch[8];
GVL.lb[iLb].valve_stopper[4].extended			:= G_IO.arDI[offset].Ch[9];
GVL.lb[iLb].valve_stopper[4].retracted			:= G_IO.arDI[offset].Ch[10];
GVL.lb[iLb].valve_stopper[5].extended			:= G_IO.arDI[offset].Ch[11];
GVL.lb[iLb].valve_stopper[5].retracted			:= G_IO.arDI[offset].Ch[12];
GVL.lb[iLb].photo_sensor[0]						:= G_IO.arDI[offset].Ch[13];
GVL.lb[iLb].photo_sensor[1]						:= G_IO.arDI[offset].Ch[14];
GVL.lb[iLb].photo_sensor[2]						:= G_IO.arDI[offset].Ch[15];



G_IO.arDO[offset].Ch[0]		:= GVL.lb[iLb].power_beltConv;
G_IO.arDO[offset].Ch[1]		:= GVL.lb[iLb].valve_stopper[0].retract;
G_IO.arDO[offset].Ch[2]		:= GVL.lb[iLb].valve_stopper[1].retract;
G_IO.arDO[offset].Ch[3]		:= GVL.lb[iLb].valve_stopper[2].retract;
G_IO.arDO[offset].Ch[4]		:= GVL.lb[iLb].valve_stopper[3].retract;
G_IO.arDO[offset].Ch[5]		:= GVL.lb[iLb].valve_stopper[4].retract;
G_IO.arDO[offset].Ch[6]		:= GVL.lb[iLb].valve_stopper[5].retract;

END_FUNCTION_BLOCK

// ---- POUs/FB_frIOmapping.TcPOU
FUNCTION_BLOCK FB_frIOmapping
VAR_INPUT
	iFR	: INT;
	mcAxis	: FB_MotionAxis_MC;	
	sNetID	: STRING;
	nSlaveAddr : UINT;
END_VAR
VAR_OUTPUT
END_VAR
VAR_IN_OUT
	IN_OUT	: ST_MotionAxis_MC;
END_VAR
VAR
	offset	: INT;
END_VAR

offset:= 75+iFR;

GVL.fr[iFR].contactor_axis	:= G_IO.arDI[offset].Ch[0];
GVL.fr[iFR].limit_sensor[0]	:= G_IO.arDI[offset].Ch[1];
GVL.fr[iFR].limit_sensor[1]	:= G_IO.arDI[offset].Ch[2];
GVL.fr[iFR].limit_sensor[2]	:= G_IO.arDI[offset].Ch[3];
GVL.fr[iFR].valve.extended	:= G_IO.arDI[offset].Ch[4];
GVL.fr[iFR].valve.retracted	:= G_IO.arDI[offset].Ch[5];

G_IO.arDO[offset].Ch[0]		:= GVL.fr[iFR].power_axis;	
G_IO.arDO[offset].Ch[1]		:= GVL.fr[iFR].valve.extend;	


mcAxis
(
	ZSN		:= GVL.fr[iFR].limit_sensor[2]	 OR IN_OUT.xHoming,
	ZSP		:= GVL.fr[iFR].limit_sensor[1]		OR IN_OUT.xHoming,
	IN_OUT	:= IN_OUT, 
	AXIS	:= GVL.fr[iFR].AxisRef, 
);
IN_OUT.bPosSensorShow	:= TRUE;
IN_OUT.bNegSensorShow	:= TRUE;
IN_OUT.bStopButtonShow	:= TRUE;
IN_OUT.rMaxAcceleration	:= 50000;
IN_OUT.rMaxDeceleration	:= 50000;
IN_OUT.rMaxJerk			:= 500000;
IN_OUT.rAcceleration	:= 2500;
IN_OUT.rDeceleration	:= 2500;
IN_OUT.rJerk			:= 12500;
IN_OUT.rMaxVelocity		:= 100;
IN_OUT.rMaxDistance		:= 50;
IN_OUT.bPosSen	:= GVL.fr[iFR].limit_sensor[1] ;
IN_OUT.bNegSen	:= GVL.fr[iFR].limit_sensor[2] ;
IN_OUT.mcHome.bCalibrationCam	:= GVL.fr[iFR].limit_sensor[0];
IN_OUT.bPositionSensor	:= GVL.fr[iFR].limit_sensor[0];
IN_OUT.bdirFW	:= TRUE;
IN_OUT.rSetPos	:= 0;
IN_OUT.sNetID := sNetID;
IN_OUT.nSlaveAddr	:= nSlaveAddr;
IN_OUT.rActTorque	:= GVL.fr_actTorque[iFR];
IN_OUT.rToqueLimitSet	:= GVL.fr_torqueLimitSet[iFR];

END_FUNCTION_BLOCK

// ---- GVLs/kitting deca/FB_valve.TcPOU
FUNCTION_BLOCK FB_valve
VAR_INPUT
	bStart	: BOOL;
	bStop	: BOOL;
END_VAR
VAR_IN_OUT
	in_out	: Valve;
END_VAR
VAR_OUTPUT
END_VAR
VAR
	rTrig_start	: R_TRIG;
	rTrig_stop	: R_TRIG;
	iState: INT;
	ton_delay	: TON;
END_VAR

rTrig_start(CLK:=bStart);
rTrig_stop(CLK:=bStop);
ton_delay(PT:=T#1S);
IF rTrig_start.Q THEN 
	iState	:= 1;
END_IF
IF rTrig_stop.Q THEN 
	iState	:= 10;
END_IF

CASE iState	OF
	0:
		;
	1:
		ton_delay.IN	:= FALSE;
		in_out.extend	:= FALSE;
		in_out.retract 	:= TRUE;
		IF in_out.retracted THEN
			iState	:= 2;
		END_IF
	2:
		ton_delay.IN	:= TRUE;
		IF ton_delay.Q THEN
			iState	:= 3;
		END_IF
	3:
		ton_delay.IN	:= FALSE;
		in_out.extend	:= TRUE;
		in_out.retract 	:= FALSE;
		IF in_out.extended THEN
			iState	:= 4;
		END_IF
	4: 
		ton_delay.IN	:= TRUE;
		IF ton_delay.Q THEN
			iState	:= 1;
		END_IF			
	10:
		in_out.extend	:= FALSE;
		in_out.retract 	:= FALSE;
		iState	:= 0;	
END_CASE

END_FUNCTION_BLOCK

// ---- GlobalTextList.TcGTLO
TEXTLIST GlobalTextList
  282 = ''
  206 = '%.2f mm'
  740 = '%.3f mm'
  386 = '%d'
  201 = '%s'
  646 = '%t'
  209 = '+'
  210 = '-'
  153 = '1'
  531 = '11111111111'
  613 = '2'
  265 = '222222'
  171 = '560-2710N/P'
  381 = 'aboveFixture_light_curtain'
  602 = 'Acc'
  843 = 'Actual Position'
  998 = 'air pressure'
  667 = 'axis'
  203 = 'Axis Error '
  89 = 'Belt'
  1107 = 'belt'
  144 = 'Belt Out'
  633 = 'belt test'
  117 = 'Belt test'
  411 = 'Belt Test'
  476 = 'belt[0]'
  143 = 'belt[1]'
  1145 = 'belt[2]'
  1131 = 'Belt_out'
  388 = 'Breaker'
  808 = 'Breaker OFF'
  486 = 'Breaker ON'
  994 = 'buffer0'
  1091 = 'Buffer0'
  1220 = 'buffer1'
  506 = 'Buffer1'
  183 = 'Buffer[0]'
  1331 = 'Buffer[1]'
  360 = 'buffer_surface_LC_slot_0'
  733 = 'button'
  235 = 'button lamp'
  856 = 'Clear'
  393 = 'cmd'
  981 = 'count'
  349 = 'Dec'
  216 = 'deg/s'
  217 = 'deg/s²'
  662 = 'DOG'
  396 = 'elapse time'
  673 = 'error'
  924 = 'Extend'
  614 = 'extended'
  781 = 'fixture clamp'
  625 = 'FR test'
  174 = 'FR Test'
  1488 = 'FR0'
  251 = 'FR1'
  1075 = 'freq'
  1168 = 'FR_axis'
  433 = 'FR_IO'
  841 = 'HOME'
  248 = 'HomeDone'
  986 = 'Infeed[0]'
  112 = 'Infeed[1]'
  886 = 'infeed[].photo_sensor[0]'
  1022 = 'inner_conveyor'
  99 = 'Jerk'
  839 = 'JOG BW'
  840 = 'JOG FW'
  1019 = 'LB'
  557 = 'LB0'
  1635 = 'LB1'
  1826 = 'LC0'
  975 = 'LC0_axis'
  253 = 'LC1'
  1342 = 'LC1_axis'
  79 = 'LCS0307-E15'
  408 = 'LC_axis'
  1539 = 'LC_IO'
  250 = 'Lift0'
  698 = 'Lift1'
  382 = 'Lift[0]'
  688 = 'Lift[1]'
  1012 = 'locked'
  373 = 'magnet'
  896 = 'magnet locked'
  447 = 'MAIN.iCnt1'
  456 = 'MAIN.tCnt1'
  492 = 'measuring light curtain'
  215 = 'mm/s'
  214 = 'mm/s²'
  207 = 'MOVE ABS'
  569 = 'Move relative'
  524 = 'ms'
  169 = 'NC_contactor'
  205 = 'Neg LS'
  749 = 'Other'
  869 = 'Others'
  530 = 'outer_conveyor'
  162 = 'Outfeed[0]'
  990 = 'Outfeed[1]'
  494 = 'outter_conveyor'
  223 = 'page1'
  737 = 'page2'
  102 = 'perturbation[0]'
  1439 = 'photo_sensor'
  70 = 'photo_sensor[0]'
  865 = 'photo_sensor[1]'
  895 = 'photo_sensor[2]'
  876 = 'PM'
  413 = 'PM0'
  1418 = 'PM1'
  809 = 'PM2'
  1129 = 'PM3'
  1328 = 'PM4'
  55 = 'PM5'
  859 = 'PM6'
  1156 = 'PM7'
  1732 = 'PM8'
  989 = 'PM9'
  1105 = 'PM_0'
  617 = 'PM_1'
  911 = 'PM_IO'
  204 = 'Pos LS'
  218 = 'power'
  844 = 'Power \nOn'
  359 = 'Power On'
  1449 = 'Power ON'
  755 = 'ReM'
  457 = 'ReM0'
  355 = 'rem0IO_0'
  452 = 'rem0IO_1'
  315 = 'rem0_IO_0'
  86 = 'rem0_IO_1'
  852 = 'ReM1'
  296 = 'ReM2'
  1185 = 'ReM3'
  904 = 'ReM4'
  274 = 'ReM5'
  882 = 'ReM6'
  996 = 'ReM7'
  763 = 'ReM8'
  1106 = 'ReM9'
  1355 = 'ReMIO_0'
  1011 = 'ReMIO_1'
  672 = 'rem_0'
  155 = 'ReM_0'
  88 = 'rem_1'
  795 = 'ReM_1'
  462 = 'Replenishment'
  199 = 'Reset'
  231 = 'RESET'
  481 = 'Retract'
  1651 = 'retract'
  934 = 'retracted'
  1226 = 'RFID[0]'
  453 = 'RFID[1]'
  186 = 'robot'
  72 = 'roller'
  81 = 'Roller IN'
  1437 = 'Roller In'
  1787 = 'Roller OUT'
  1125 = 'Roller Out'
  499 = 'Servo'
  983 = 'Set absolute\nencoder as line'
  622 = 'Set absolute\nencoder as linear'
  454 = 'Set absolute\nencoder as rotation'
  606 = 'Set absolute \nencoder as line'
  230 = 'Set absolute encoder\n'
  976 = 'Set absoluteencoder \nas line'
  545 = 'Set Incremental encoder'
  883 = 'Set incremental encoder'
  871 = 'Set incremental encoder \nas line'
  719 = 'Set incremental encoder as line'
  208 = 'Set Point'
  14 = 'Set Pos to 0'
  284 = 'sick measure'
  765 = 'SLC'
  971 = 'slot_0'
  156 = 'slot_1'
  122 = 'slot_2'
  1494 = 'START'
  198 = 'Stop'
  399 = 'STOP'
  336 = 'surface_light_curtain'
  379 = 'time'
  1753 = 'valve'
  637 = 'valve_clamp'
  863 = 'valve_clamp[0]'
  712 = 'valve_clamp[1]'
  739 = 'valve_expand'
  1456 = 'valve_guide[0]'
  1699 = 'valve_guide[1]'
  1384 = 'valve_inner[0]'
  67 = 'valve_inner[1]'
  1359 = 'valve_inner[2]'
  668 = 'valve_lift'
  1180 = 'valve_outer[0]'
  1288 = 'valve_outer[1]'
  728 = 'valve_outter[0]'
  516 = 'valve_perturbation[0]'
  836 = 'valve_perturbation[1]'
  970 = 'valve_perturbation[2]'
  148 = 'valve_perturbation[3]'
  227 = 'valve_stopper'
  192 = 'valve_stopper[0]'
  1065 = 'valve_stopper[1]'
  1212 = 'valve_stopper[2]'
  1778 = 'valve_stopper[3]'
  1546 = 'valve_stopper[4]'
  1487 = 'valve_stopper[5]'
  200 = 'Velocity'
  794 = 'Write'
  729 = 'Write '
  403 = 'X'
  404 = 'Y'
  405 = 'Z'
  607 = '计数'
  641 = '计算'
  664 = '页面1'
END_TEXTLIST

